KUKA KRL program: MyProgram_095().src

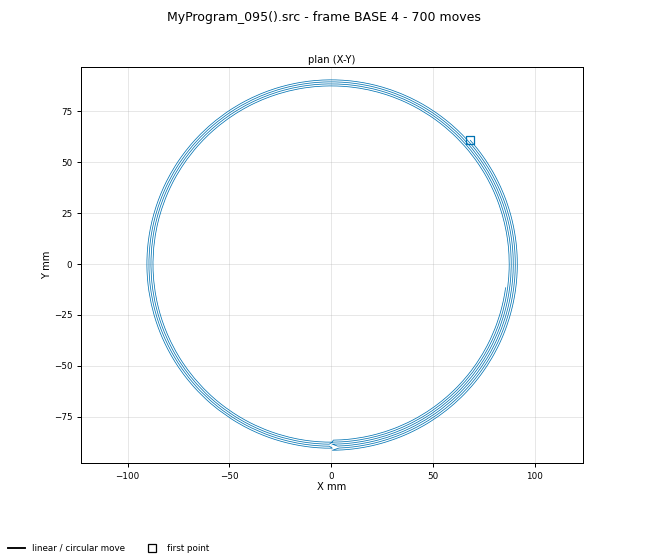
[picture p0: tool path of MyProgram_095().src in frame BASE 4, 700 of 700 moves have a stored position in this frame; points joined in program order, loops and branches not executed]
&ACCESS RVP
&REL 1
&PARAM TEMPLATE = C:\KRC\Roboter\Template\vorgabe
&PARAM EDITMASK = *
DEF MyProgram_095()
; ---- Setting reference (Base) ----
$BASE = BASE_DATA[4]

; --------------------------
; ---- Setting tool (TCP) ----
$TOOL = TOOL_DATA[3]
; --------------------------

$VEL.CP = VEL_APROX_PRINT
Startdeposition()
$VEL.CP = VEL_PRINT
LIN {X 68.4348,Y 60.7863,Z 89,A 36.1142,B 24.9115,C -2.1728,E1 25.1202,E2 408.9447} C_DIS
LIN {X 69.906,Y 59.0885,Z 89,A 34.5968,B 24.912,C -2.1656,E1 25.123,E2 410.4721} C_DIS
LIN {X 71.8852,Y 56.6631,Z 89,A 32.7208,B 24.9122,C -2.1639,E1 25.1263,E2 412.3433} C_DIS
LIN {X 73.5209,Y 54.5268,Z 89,A 31.0903,B 24.9124,C -2.1617,E1 25.129,E2 413.9712} C_DIS
LIN {X 74.8369,Y 52.7061,Z 89,A 29.6918,B 24.9126,C -2.1585,E1 25.1313,E2 415.3706} C_DIS
LIN {X 76.1078,Y 50.8536,Z 89,A 28.2935,B 24.9129,C -2.1552,E1 25.1335,E2 416.7698} C_DIS
LIN {X 77.3329,Y 48.9705,Z 89,A 26.8951,B 24.9132,C -2.1518,E1 25.1356,E2 418.169} C_DIS
LIN {X 78.5114,Y 47.0579,Z 89,A 25.4966,B 24.9134,C -2.1484,E1 25.1376,E2 419.5685} C_DIS
LIN {X 79.5405,Y 45.2947,Z 89,A 24.2263,B 24.9137,C -2.1453,E1 25.1394,E2 420.8396} C_DIS
LIN {X 80.6281,Y 43.329,Z 89,A 22.8286,B 24.914,C -2.1418,E1 25.1413,E2 422.2383} C_DIS
LIN {X 81.9545,Y 40.7633,Z 89,A 20.9127,B 24.9147,C -2.1329,E1 25.1437,E2 424.165} C_DIS
LIN {X 83.2199,Y 38.1175,Z 89,A 19.2069,B 24.9147,C -2.1324,E1 25.1457,E2 425.8628} C_DIS
LIN {X 84.1302,Y 36.0637,Z 89,A 17.8095,B 24.915,C -2.1287,E1 25.1473,E2 427.2613} C_DIS
LIN {X 84.9127,Y 34.178,Z 89,A 16.5212,B 24.9153,C -2.1247,E1 25.1486,E2 428.552} C_DIS
LIN {X 86.1131,Y 31.0294,Z 89,A 14.4253,B 24.9158,C -2.119,E1 25.1507,E2 430.6496} C_DIS
LIN {X 86.9142,Y 28.7126,Z 89,A 12.9188,B 24.9161,C -2.1154,E1 25.152,E2 432.1561} C_DIS
LIN {X 87.532,Y 26.7667,Z 89,A 11.6496,B 24.9164,C -2.1119,E1 25.1531,E2 433.4263} C_DIS
LIN {X 88.3281,Y 24.0072,Z 89,A 9.739,B 24.9171,C -2.1024,E1 25.1545,E2 435.3484} C_DIS
LIN {X 89.0572,Y 21.1497,Z 89,A 8.0298,B 24.9171,C -2.1017,E1 25.1557,E2 437.0493} C_DIS
LIN {X 89.6843,Y 18.3008,Z 89,A 6.1409,B 24.9178,C -2.0938,E1 25.1568,E2 438.9459} C_DIS
LIN {X 90.2812,Y 15.0822,Z 89,A 4.0769,B 24.9183,C -2.0868,E1 25.1578,E2 441.0142} C_DIS
LIN {X 90.6725,Y 12.5216,Z 89,A 2.552,B 24.9185,C -2.0853,E1 25.1584,E2 442.5338} C_DIS
LIN {X 90.9525,Y 10.2926,Z 89,A 1.1555,B 24.9188,C -2.0812,E1 25.1589,E2 443.9317} C_DIS
LIN {X 91.2533,Y 7.1433,Z 89,A -0.8295,B 24.9193,C -2.0747,E1 25.1594,E2 445.9201} C_DIS
LIN {X 91.4238,Y 4.4914,Z 89,A -2.4448,B 24.9196,C -2.0712,E1 25.1596,E2 447.5343} C_DIS
LIN {X 91.5002,Y 2.4512,Z 89,A -3.8938,B 24.9204,C -2.0608,E1 25.1598,E2 448.999} C_DIS
LIN {X 91.5272,Y -1.1233,Z 89,A -5.9356,B 24.9204,C -2.0608,E1 25.1598,E2 451.0288} C_DIS
LIN {X 91.4721,Y -3.3691,Z 89,A -7.3323,B 24.9207,C -2.0566,E1 25.1596,E2 452.427} C_DIS
LIN {X 91.2861,Y -6.7337,Z 89,A -9.4265,B 24.9212,C -2.0504,E1 25.1593,E2 454.5234} C_DIS
LIN {X 91.0357,Y -9.5222,Z 89,A -11.2776,B 24.9219,C -2.0412,E1 25.1588,E2 456.3854} C_DIS
LIN {X 90.7277,Y -12.1155,Z 89,A -12.8086,B 24.9219,C -2.0397,E1 25.1583,E2 457.9108} C_DIS
LIN {X 90.403,Y -14.3384,Z 89,A -14.205,B 24.9223,C -2.0356,E1 25.1577,E2 459.3087} C_DIS
LIN {X 90.0239,Y -16.5527,Z 89,A -15.583,B 24.9226,C -2.0321,E1 25.157,E2 460.6868} C_DIS
LIN {X 89.5906,Y -18.757,Z 89,A -16.9981,B 24.9229,C -2.0273,E1 25.1562,E2 462.1049} C_DIS
LIN {X 89.1033,Y -20.95,Z 89,A -18.3945,B 24.9232,C -2.0232,E1 25.1553,E2 463.503} C_DIS
LIN {X 88.3471,Y -23.9366,Z 89,A -20.3496,B 24.9238,C -2.0162,E1 25.154,E2 465.4634} C_DIS
LIN {X 87.5927,Y -26.5709,Z 89,A -21.9951,B 24.924,C -2.0133,E1 25.1527,E2 467.1063} C_DIS
LIN {X 86.9773,Y -28.5176,Z 89,A -23.2641,B 24.9243,C -2.0097,E1 25.1516,E2 468.3767} C_DIS
LIN {X 86.2512,Y -30.6435,Z 89,A -24.6609,B 24.9246,C -2.0057,E1 25.1503,E2 469.7751} C_DIS
LIN {X 85.5341,Y -32.5902,Z 89,A -26.0056,B 24.925,C -2,E1 25.149,E2 471.1257} C_DIS
LIN {X 84.6437,Y -34.8388,Z 89,A -27.4729,B 24.9252,C -1.997,E1 25.1474,E2 472.5918} C_DIS
LIN {X 83.7633,Y -36.9055,Z 89,A -28.8517,B 24.9255,C -1.9938,E1 25.1459,E2 473.9708} C_DIS
LIN {X 82.8323,Y -38.9501,Z 89,A -30.2672,B 24.9258,C -1.9892,E1 25.1442,E2 475.3893} C_DIS
LIN {X 81.7605,Y -41.1548,Z 89,A -31.9887,B 24.9267,C -1.9778,E1 25.1421,E2 477.1286} C_DIS
LIN {X 80.1903,Y -44.1362,Z 89,A -33.8687,B 24.9265,C -1.98,E1 25.1396,E2 478.9936} C_DIS
LIN {X 79.083,Y -46.0909,Z 89,A -35.2665,B 24.9268,C -1.9762,E1 25.1377,E2 480.393} C_DIS
LIN {X 77.928,Y -48.0178,Z 89,A -36.6636,B 24.927,C -1.9725,E1 25.1356,E2 481.7917} C_DIS
LIN {X 76.7342,Y -49.9032,Z 89,A -38.0524,B 24.9273,C -1.9689,E1 25.1335,E2 483.1821} C_DIS
LIN {X 75.2678,Y -52.0862,Z 89,A -39.8077,B 24.9279,C -1.9604,E1 25.1308,E2 484.9489} C_DIS
LIN {X 73.5209,Y -54.5268,Z 89,A -41.556,B 24.9279,C -1.96,E1 25.1279,E2 486.6897} C_DIS
LIN {X 72.2857,Y -56.1523,Z 89,A -42.8446,B 24.9283,C -1.9562,E1 25.1257,E2 487.9811} C_DIS
LIN {X 70.7568,Y -58.0686,Z 89,A -44.3521,B 24.9285,C -1.9531,E1 25.1231,E2 489.4889} C_DIS
LIN {X 69.3104,Y -59.7876,Z 89,A -45.7504,B 24.9287,C -1.9497,E1 25.1205,E2 490.8888} C_DIS
LIN {X 67.0628,Y -62.2982,Z 89,A -47.8483,B 24.9291,C -1.9448,E1 25.1166,E2 492.989} C_DIS
LIN {X 65.5138,Y -63.9252,Z 89,A -49.2469,B 24.9293,C -1.9416,E1 25.1139,E2 494.3892} C_DIS
LIN {X 63.9252,Y -65.5138,Z 89,A -50.6456,B 24.9295,C -1.9385,E1 25.1111,E2 495.7893} C_DIS
LIN {X 62.2982,Y -67.0628,Z 89,A -52.0445,B 24.9298,C -1.9354,E1 25.1083,E2 497.1897} C_DIS
LIN {X 60.7039,Y -68.5086,Z 89,A -53.59,B 24.9305,C -1.9252,E1 25.105,E2 498.7532} C_DIS
LIN {X 58.2262,Y -70.6258,Z 89,A -55.415,B 24.9303,C -1.9284,E1 25.1011,E2 500.5637} C_DIS
LIN {X 56.4754,Y -72.0335,Z 89,A -56.833,B 24.9305,C -1.9249,E1 25.098,E2 501.9846} C_DIS
LIN {X 54.6906,Y -73.3978,Z 89,A -58.2143,B 24.9307,C -1.9228,E1 25.0949,E2 503.3659} C_DIS
LIN {X 53.0381,Y -74.6,Z 89,A -59.5276,B 24.931,C -1.919,E1 25.092,E2 504.6836} C_DIS
LIN {X 50.8536,Y -76.1078,Z 89,A -61.142,B 24.931,C -1.9173,E1 25.0882,E2 506.2965} C_DIS
LIN {X 49.143,Y -77.2222,Z 89,A -62.4148,B 24.9312,C -1.915,E1 25.0852,E2 507.5706} C_DIS
LIN {X 47.2331,Y -78.405,Z 89,A -63.8151,B 24.9314,C -1.9126,E1 25.0819,E2 508.9721} C_DIS
LIN {X 45.2947,Y -79.5405,Z 89,A -65.2344,B 24.9316,C -1.9096,E1 25.0785,E2 510.3943} C_DIS
LIN {X 42.4309,Y -81.104,Z 89,A -67.2665,B 24.9319,C -1.9065,E1 25.0735,E2 512.428} C_DIS
LIN {X 40.332,Y -82.1683,Z 89,A -68.7183,B 24.9319,C -1.9048,E1 25.0698,E2 513.8798} C_DIS
LIN {X 38.1175,Y -83.2199,Z 89,A -70.2478,B 24.9321,C -1.9025,E1 25.066,E2 515.4108} C_DIS
LIN {X 36.0637,Y -84.1302,Z 89,A -71.6494,B 24.9323,C -1.9006,E1 25.0624,E2 516.8135} C_DIS
LIN {X 33.9882,Y -84.99,Z 89,A -73.247,B 24.9329,C -1.8919,E1 25.0582,E2 518.428} C_DIS
LIN {X 30.8369,Y -86.1834,Z 89,A -75.1546,B 24.9326,C -1.8961,E1 25.0532,E2 520.3216} C_DIS
LIN {X 28.7126,Y -86.9142,Z 89,A -76.5571,B 24.9327,C -1.8945,E1 25.0495,E2 521.7252} C_DIS
LIN {X 26.7667,Y -87.532,Z 89,A -77.8313,B 24.9328,C -1.8932,E1 25.0461,E2 523.0004} C_DIS
LIN {X 24.4133,Y -88.2184,Z 89,A -79.3626,B 24.9329,C -1.8916,E1 25.042,E2 524.5328} C_DIS
LIN {X 22.241,Y -88.7909,Z 89,A -80.7653,B 24.933,C -1.8903,E1 25.0382,E2 525.9364} C_DIS
LIN {X 20.0552,Y -89.31,Z 89,A -82.1687,B 24.9331,C -1.889,E1 25.0344,E2 527.3409} C_DIS
LIN {X 17.8574,Y -89.7753,Z 89,A -83.5725,B 24.9331,C -1.8879,E1 25.0305,E2 528.7457} C_DIS
LIN {X 15.6488,Y -90.1865,Z 89,A -85.1605,B 24.9337,C -1.8806,E1 25.0261,E2 530.3492} C_DIS
LIN {X 12.5216,Y -90.6725,Z 89,A -86.9727,B 24.9334,C -1.8849,E1 25.0212,E2 532.1494} C_DIS
LIN {X 10.2926,Y -90.9525,Z 89,A -88.377,B 24.9334,C -1.8841,E1 25.0173,E2 533.5545} C_DIS
LIN {X 8.0575,Y -91.1777,Z 89,A -89.7817,B 24.9335,C -1.8835,E1 25.0134,E2 534.9601} C_DIS
LIN {X 5.8174,Y -91.348,Z 89,A -91.1865,B 24.9335,C -1.8829,E1 25.0094,E2 536.3656} C_DIS
LIN {X 2.5555,Y -91.497,Z 89,A -93.2493,B 24.9336,C -1.8815,E1 25.0037,E2 538.4311} C_DIS
LIN {X 0.6147,Y -91.5303,Z 89,A -94.1302,B 24.9329,C -1.8925,E1 25.0013,E2 539.2859} C_DIS
Enddeposition()
LIN {X 0.6147,Y -91.5303,Z 89,A -94.1302,B 24.9329,C -1.8925,E1 25.0013,E2 539.2859} C_DIS
Startdeposition()
$VEL.CP = VEL_PRINT
LIN {X 3.841,Y -90.4576,Z 89,A -91.6476,B 24.9305,C -1.9253,E1 25.0084,E2 536.7259} C_DIS
LIN {X 6.8274,Y -90.2822,Z 89,A -89.6587,B 24.9302,C -1.9294,E1 25.014,E2 534.7283} C_DIS
LIN {X 10.5822,Y -89.9186,Z 89,A -87.3173,B 24.9302,C -1.9292,E1 25.0205,E2 532.3889} C_DIS
LIN {X 13.8939,Y -89.4668,Z 89,A -84.9684,B 24.9295,C -1.9387,E1 25.027,E2 530.0197} C_DIS
LIN {X 18.0628,Y -88.7192,Z 89,A -82.5559,B 24.93,C -1.9317,E1 25.0336,E2 527.6266} C_DIS
LIN {X 21.585,Y -87.9286,Z 89,A -80.3322,B 24.93,C -1.9317,E1 25.0397,E2 525.4058} C_DIS
LIN {X 23.7624,Y -87.3654,Z 89,A -78.7831,B 24.9296,C -1.9376,E1 25.0439,E2 523.8453} C_DIS
LIN {X 27.8255,Y -86.1573,Z 89,A -75.9416,B 24.929,C -1.9463,E1 25.0515,E2 520.9884} C_DIS
LIN {X 32.3644,Y -84.5576,Z 89,A -72.9807,B 24.929,C -1.9473,E1 25.0592,E2 518.0312} C_DIS
LIN {X 36.0562,Y -83.05,Z 89,A -70.5763,B 24.929,C -1.9468,E1 25.0654,E2 515.6336} C_DIS
LIN {X 39.4601,Y -81.4881,Z 89,A -68.247,B 24.9288,C -1.9491,E1 25.0713,E2 513.3049} C_DIS
LIN {X 42.1763,Y -80.1155,Z 89,A -65.821,B 24.9272,C -1.9701,E1 25.0774,E2 510.8361} C_DIS
LIN {X 45.1686,Y -78.4674,Z 89,A -64.2021,B 24.9284,C -1.9546,E1 25.0812,E2 509.2585} C_DIS
LIN {X 48.0241,Y -76.753,Z 89,A -61.7848,B 24.9273,C -1.9696,E1 25.087,E2 506.8135} C_DIS
LIN {X 51.7728,Y -74.276,Z 89,A -59.1835,B 24.9275,C -1.9666,E1 25.093,E2 504.2281} C_DIS
LIN {X 53.7404,Y -72.8657,Z 89,A -57.2283,B 24.9261,C -1.985,E1 25.0975,E2 502.2365} C_DIS
LIN {X 56.4119,Y -70.8178,Z 89,A -55.1326,B 24.9259,C -1.9884,E1 25.102,E2 500.1406} C_DIS
LIN {X 58.9229,Y -68.7422,Z 89,A -53.6408,B 24.9271,C -1.9725,E1 25.1051,E2 498.6921} C_DIS
LIN {X 60.8149,Y -67.075,Z 89,A -51.7631,B 24.926,C -1.9863,E1 25.1091,E2 496.7893} C_DIS
LIN {X 63.9525,Y -64.0907,Z 89,A -49.1215,B 24.9258,C -1.9893,E1 25.1144,E2 494.1516} C_DIS
LIN {X 66.8951,Y -61.0119,Z 89,A -46.6842,B 24.926,C -1.9867,E1 25.119,E2 491.7311} C_DIS
LIN {X 68.7114,Y -58.9592,Z 89,A -44.8258,B 24.9253,C -1.9957,E1 25.1224,E2 489.86} C_DIS
LIN {X 70.8722,Y -56.343,Z 89,A -42.7154,B 24.925,C -2,E1 25.1261,E2 487.7491} C_DIS
LIN {X 72.9495,Y -53.6259,Z 89,A -40.3766,B 24.9241,C -2.0122,E1 25.1301,E2 485.3927} C_DIS
LIN {X 74.6947,Y -51.1692,Z 89,A -38.0119,B 24.9224,C -2.0342,E1 25.1339,E2 482.9877} C_DIS
LIN {X 76.7688,Y -47.9989,Z 89,A -36.3079,B 24.9238,C -2.0156,E1 25.1363,E2 481.3363} C_DIS
LIN {X 78.8273,Y -44.5399,Z 89,A -33.7021,B 24.9231,C -2.025,E1 25.14,E2 478.7215} C_DIS
LIN {X 80.3925,Y -41.6488,Z 89,A -31.6323,B 24.9227,C -2.0308,E1 25.1427,E2 476.6491} C_DIS
LIN {X 81.849,Y -38.7087,Z 89,A -29.5508,B 24.9222,C -2.0371,E1 25.1452,E2 474.5638} C_DIS
LIN {X 83.2517,Y -35.5907,Z 89,A -27.6678,B 24.9225,C -2.0334,E1 25.1473,E2 472.6998} C_DIS
LIN {X 84.5175,Y -32.4701,Z 89,A -25.045,B 24.9206,C -2.058,E1 25.15,E2 470.0335} C_DIS
LIN {X 85.8563,Y -28.7415,Z 89,A -22.8423,B 24.9208,C -2.0546,E1 25.152,E2 467.8513} C_DIS
LIN {X 86.8313,Y -25.645,Z 89,A -20.7763,B 24.9203,C -2.0614,E1 25.1537,E2 465.7809} C_DIS
LIN {X 87.7136,Y -22.4425,Z 89,A -18.7465,B 24.92,C -2.0654,E1 25.1552,E2 463.7534} C_DIS
LIN {X 88.4899,Y -19.1544,Z 89,A -16.7256,B 24.9198,C -2.0679,E1 25.1564,E2 461.7384} C_DIS
LIN {X 89.1025,Y -16.0649,Z 89,A -14.6764,B 24.9192,C -2.0763,E1 25.1575,E2 459.6813} C_DIS
LIN {X 89.7875,Y -11.642,Z 89,A -11.4066,B 24.9172,C -2.1015,E1 25.1588,E2 456.3713} C_DIS
LIN {X 90.2839,Y -6.8065,Z 89,A -8.9059,B 24.9181,C -2.0901,E1 25.1594,E2 453.9122} C_DIS
LIN {X 90.4532,Y -3.9434,Z 89,A -7.0295,B 24.9174,C -2.0982,E1 25.1597,E2 452.0278} C_DIS
LIN {X 90.5369,Y -0.7324,Z 89,A -4.9658,B 24.9168,C -2.1059,E1 25.1597,E2 449.9584} C_DIS
LIN {X 90.4983,Y 2.7184,Z 89,A -2.7827,B 24.9163,C -2.1129,E1 25.1597,E2 447.7718} C_DIS
LIN {X 90.3216,Y 6.2745,Z 89,A -0.5065,B 24.9156,C -2.1209,E1 25.1593,E2 445.4902} C_DIS
LIN {X 90.012,Y 9.7618,Z 89,A 1.5203,B 24.9156,C -2.1209,E1 25.1587,E2 443.4751} C_DIS
LIN {X 89.7383,Y 12.0216,Z 89,A 3.2086,B 24.9145,C -2.1346,E1 25.1581,E2 441.7648} C_DIS
LIN {X 89.1963,Y 15.5434,Z 89,A 5.1496,B 24.9149,C -2.1301,E1 25.1573,E2 439.8457} C_DIS
LIN {X 88.7451,Y 17.9364,Z 89,A 6.8451,B 24.9141,C -2.1406,E1 25.1563,E2 438.1354} C_DIS
LIN {X 88.0369,Y 21.141,Z 89,A 8.9727,B 24.9134,C -2.1488,E1 25.155,E2 436.0007} C_DIS
LIN {X 87.4365,Y 23.4992,Z 89,A 10.4329,B 24.9133,C -2.1506,E1 25.154,E2 434.5447} C_DIS
LIN {X 85.8607,Y 28.7284,Z 89,A 13.9051,B 24.9124,C -2.1615,E1 25.1511,E2 431.0665} C_DIS
LIN {X 84.6865,Y 32.024,Z 89,A 15.7904,B 24.9128,C -2.1561,E1 25.1493,E2 429.2045} C_DIS
LIN {X 83.1699,Y 35.7813,Z 89,A 18.5222,B 24.9117,C -2.1695,E1 25.1464,E2 426.4561} C_DIS
LIN {X 82.0179,Y 38.3461,Z 89,A 20.4762,B 24.9108,C -2.1809,E1 25.1441,E2 424.4859} C_DIS
LIN {X 80.8031,Y 40.8455,Z 89,A 22.4831,B 24.9096,C -2.1947,E1 25.1416,E2 422.4569} C_DIS
LIN {X 78.9088,Y 44.3939,Z 89,A 24.6853,B 24.9101,C -2.1892,E1 25.1386,E2 420.2793} C_DIS
LIN {X 77.2267,Y 47.2594,Z 89,A 26.4874,B 24.9105,C -2.184,E1 25.1361,E2 418.4987} C_DIS
LIN {X 75.5281,Y 49.9285,Z 89,A 28.8052,B 24.9092,C -2.2004,E1 25.1325,E2 416.1537} C_DIS
LIN {X 73.3795,Y 53.0386,Z 89,A 31.4469,B 24.9079,C -2.2153,E1 25.1282,E2 413.4897} C_DIS
LIN {X 70.8403,Y 56.3833,Z 89,A 33.677,B 24.9087,C -2.2065,E1 25.1244,E2 411.2911} C_DIS
LIN {X 69.0223,Y 58.5942,Z 89,A 35.5338,B 24.9082,C -2.2123,E1 25.1211,E2 409.4289} C_DIS
LIN {X 66.3294,Y 61.6273,Z 89,A 37.9615,B 24.9082,C -2.2131,E1 25.1166,E2 407.0102} C_DIS
LIN {X 64.3928,Y 63.6467,Z 89,A 39.855,B 24.9074,C -2.2213,E1 25.1129,E2 405.1055} C_DIS
LIN {X 61.9374,Y 66.0387,Z 89,A 41.718,B 24.908,C -2.215,E1 25.1092,E2 403.265} C_DIS
LIN {X 59.5402,Y 68.2078,Z 89,A 44.0276,B 24.9069,C -2.2283,E1 25.1043,E2 400.9333} C_DIS
LIN {X 57.492,Y 69.9446,Z 89,A 45.8102,B 24.9063,C -2.2344,E1 25.1005,E2 399.1431} C_DIS
LIN {X 54.2039,Y 72.5212,Z 89,A 48.5095,B 24.9058,C -2.2411,E1 25.0945,E2 396.4377} C_DIS
LIN {X 51.4181,Y 74.5226,Z 89,A 50.2979,B 24.9066,C -2.2315,E1 25.0905,E2 394.6783} C_DIS
LIN {X 47.9538,Y 76.797,Z 89,A 53.2119,B 24.9054,C -2.2457,E1 25.0836,E2 391.7403} C_DIS
LIN {X 45.0435,Y 78.5393,Z 89,A 55.3345,B 24.9052,C -2.2479,E1 25.0785,E2 389.6188} C_DIS
LIN {X 42.687,Y 79.8461,Z 89,A 57.3502,B 24.9041,C -2.2609,E1 25.0735,E2 387.578} C_DIS
LIN {X 38.919,Y 81.7481,Z 89,A 59.8208,B 24.9044,C -2.2573,E1 25.0673,E2 385.1226} C_DIS
LIN {X 34.2257,Y 83.8209,Z 89,A 63.3531,B 24.9033,C -2.2706,E1 25.0582,E2 381.5673} C_DIS
LIN {X 29.4174,Y 85.6284,Z 89,A 66.5241,B 24.9033,C -2.2707,E1 25.0499,E2 378.4024} C_DIS
LIN {X 25.2199,Y 86.957,Z 89,A 69.0295,B 24.9039,C -2.2632,E1 25.0432,E2 375.9192} C_DIS
LIN {X 21.9677,Y 87.8352,Z 89,A 71.1397,B 24.9039,C -2.2638,E1 25.0375,E2 373.8109} C_DIS
LIN {X 18.9594,Y 88.5324,Z 89,A 72.9796,B 24.9041,C -2.261,E1 25.0325,E2 371.9801} C_DIS
LIN {X 15.891,Y 89.1338,Z 89,A 75.0794,B 24.9037,C -2.2658,E1 25.0267,E2 369.8712} C_DIS
LIN {X 12.4524,Y 89.6792,Z 89,A 77.0943,B 24.9042,C -2.2602,E1 25.0212,E2 367.8716} C_DIS
LIN {X 9.4502,Y 90.0446,Z 89,A 79.136,B 24.9038,C -2.2647,E1 25.0155,E2 365.8206} C_DIS
LIN {X 5.8559,Y 90.3499,Z 89,A 81.4804,B 24.9036,C -2.2669,E1 25.009,E2 363.4722} C_DIS
LIN {X 2.2826,Y 90.5117,Z 89,A 83.5521,B 24.9042,C -2.2604,E1 25.0033,E2 361.4165} C_DIS
LIN {X -0.6869,Y 90.5366,Z 89,A 85.6422,B 24.9036,C -2.2669,E1 24.9974,E2 359.3109} C_DIS
LIN {X -4.2126,Y 90.4417,Z 89,A 87.8996,B 24.9036,C -2.267,E1 24.9911,E2 357.0528} C_DIS
LIN {X -7.9472,Y 90.1905,Z 89,A 90.2515,B 24.9037,C -2.2654,E1 24.9845,E2 354.7037} C_DIS
LIN {X -11.1573,Y 89.8503,Z 89,A 92.3303,B 24.9037,C -2.2654,E1 24.9788,E2 352.6236} C_DIS
LIN {X -14.8513,Y 89.3128,Z 89,A 94.5753,B 24.9042,C -2.2601,E1 24.9726,E2 350.3893} C_DIS
LIN {X -17.601,Y 88.8122,Z 89,A 96.6821,B 24.9034,C -2.2695,E1 24.9668,E2 348.2577} C_DIS
LIN {X -21.5979,Y 87.9255,Z 89,A 99.0047,B 24.9043,C -2.2585,E1 24.9605,E2 345.9582} C_DIS
LIN {X -24.8007,Y 87.0763,Z 89,A 100.9732,B 24.9048,C -2.2523,E1 24.9552,E2 344.0015} C_DIS
LIN {X -27.4177,Y 86.2893,Z 89,A 102.8866,B 24.9045,C -2.2561,E1 24.9501,E2 342.0756} C_DIS
LIN {X -31.1882,Y 84.998,Z 89,A 105.4157,B 24.9048,C -2.2532,E1 24.9435,E2 339.5484} C_DIS
LIN {X -34.5944,Y 83.6708,Z 89,A 107.5352,B 24.9055,C -2.2439,E1 24.938,E2 337.4465} C_DIS
LIN {X -38.8381,Y 81.787,Z 89,A 110.6816,B 24.9054,C -2.246,E1 24.93,E2 334.2873} C_DIS
LIN {X -41.879,Y 80.2721,Z 89,A 112.7855,B 24.9058,C -2.2411,E1 24.9248,E2 332.1895} C_DIS
LIN {X -44.5871,Y 78.8009,Z 89,A 115.1067,B 24.9051,C -2.2493,E1 24.919,E2 329.842} C_DIS
LIN {X -48.6235,Y 76.3754,Z 89,A 117.709,B 24.9065,C -2.232,E1 24.9129,E2 327.2727} C_DIS
LIN {X -51.4688,Y 74.4874,Z 89,A 119.8592,B 24.9069,C -2.2275,E1 24.908,E2 325.1262} C_DIS
LIN {X -56.755,Y 70.543,Z 89,A 124.383,B 24.9068,C -2.2294,E1 24.8979,E2 320.5812} C_DIS
LIN {X -60.1524,Y 67.6692,Z 89,A 126.781,B 24.9084,C -2.2103,E1 24.8929,E2 318.2195} C_DIS
LIN {X -64.183,Y 63.8591,Z 89,A 130.3958,B 24.9088,C -2.2052,E1 24.8856,E2 314.6018} C_DIS
LIN {X -66.9222,Y 60.9824,Z 89,A 132.9651,B 24.9092,C -2.2007,E1 24.8807,E2 312.032} C_DIS
LIN {X -69.0691,Y 58.5393,Z 89,A 135.7258,B 24.9078,C -2.2168,E1 24.8756,E2 309.2202} C_DIS
LIN {X -71.5763,Y 55.4457,Z 89,A 137.5885,B 24.91,C -2.1902,E1 24.8725,E2 307.4124} C_DIS
LIN {X -73.5936,Y 52.7385,Z 89,A 139.6955,B 24.9106,C -2.1835,E1 24.8691,E2 305.311} C_DIS
LIN {X -75.3144,Y 50.2526,Z 89,A 141.7065,B 24.9108,C -2.1811,E1 24.8659,E2 303.2956} C_DIS
LIN {X -76.5996,Y 48.2697,Z 89,A 143.2253,B 24.9111,C -2.1777,E1 24.8636,E2 301.7774} C_DIS
LIN {X -78.7995,Y 44.5894,Z 89,A 146.1309,B 24.9112,C -2.1757,E1 24.8595,E2 298.8615} C_DIS
LIN {X -80.8397,Y 40.7739,Z 89,A 148.829,B 24.912,C -2.1664,E1 24.8561,E2 296.171} C_DIS
LIN {X -82.3206,Y 37.6953,Z 89,A 150.9163,B 24.9127,C -2.1577,E1 24.8536,E2 294.0931} C_DIS
LIN {X -83.798,Y 34.282,Z 89,A 153.1681,B 24.9135,C -2.1476,E1 24.8512,E2 291.8531} C_DIS
LIN {X -84.9131,Y 31.4209,Z 89,A 155.6055,B 24.9128,C -2.1564,E1 24.8488,E2 289.3807} C_DIS
LIN {X -85.9862,Y 28.3543,Z 89,A 157.9259,B 24.9127,C -2.158,E1 24.8468,E2 287.0433} C_DIS
LIN {X -87.1572,Y 24.5149,Z 89,A 159.6948,B 24.9152,C -2.1269,E1 24.8455,E2 285.3383} C_DIS
LIN {X -88.0666,Y 21.0193,Z 89,A 162.16,B 24.9153,C -2.1251,E1 24.8438,E2 282.8632} C_DIS
LIN {X -88.8209,Y 17.5612,Z 89,A 164.3658,B 24.916,C -2.1169,E1 24.8425,E2 280.6638} C_DIS
LIN {X -89.4048,Y 14.2946,Z 89,A 166.4804,B 24.9164,C -2.1107,E1 24.8416,E2 278.5516} C_DIS
LIN {X -89.8714,Y 10.9855,Z 89,A 168.3538,B 24.9176,C -2.0968,E1 24.8409,E2 276.7003} C_DIS
LIN {X -90.1183,Y 8.7287,Z 89,A 170.0477,B 24.9173,C -2.0998,E1 24.8404,E2 274.9889} C_DIS
LIN {X -90.3804,Y 5.3726,Z 89,A 172.1787,B 24.9178,C -2.093,E1 24.84,E2 272.8614} C_DIS
LIN {X -90.5176,Y 2.0025,Z 89,A 174.2642,B 24.9185,C -2.0847,E1 24.8398,E2 270.7831} C_DIS
LIN {X -90.5355,Y -0.9214,Z 89,A 176.0887,B 24.919,C -2.078,E1 24.8398,E2 268.9636} C_DIS
LIN {X -90.4602,Y -3.782,Z 89,A 177.956,B 24.9193,C -2.0739,E1 24.84,E2 267.0948} C_DIS
LIN {X -90.2522,Y -7.203,Z 89,A -179.8808,B 24.9199,C -2.0669,E1 24.8404,E2 264.9354} C_DIS
LIN {X -89.937,Y -10.4248,Z 89,A -178.1412,B 24.9211,C -2.0512,E1 24.8409,E2 263.2227} C_DIS
LIN {X -89.5869,Y -13.102,Z 89,A -176.1167,B 24.9208,C -2.0552,E1 24.8417,E2 261.1765} C_DIS
LIN {X -88.3611,Y -19.7448,Z 89,A -171.9405,B 24.922,C -2.039,E1 24.8439,E2 257.0145} C_DIS
LIN {X -86.9694,Y -25.1777,Z 89,A -168.234,B 24.9225,C -2.0328,E1 24.8465,E2 253.3011} C_DIS
LIN {X -86.0678,Y -28.1022,Z 89,A -166.2597,B 24.9229,C -2.0282,E1 24.8482,E2 251.3265} C_DIS
LIN {X -85.0374,Y -31.0801,Z 89,A -164.352,B 24.9235,C -2.0197,E1 24.8499,E2 249.4282} C_DIS
LIN {X -84.02,Y -33.7367,Z 89,A -162.5395,B 24.9239,C -2.0149,E1 24.8518,E2 247.6171} C_DIS
LIN {X -82.9012,Y -36.3975,Z 89,A -160.4792,B 24.9237,C -2.0167,E1 24.8541,E2 245.5409} C_DIS
LIN {X -81.6835,Y -39.0534,Z 89,A -158.7203,B 24.9243,C -2.0088,E1 24.8561,E2 243.7913} C_DIS
LIN {X -80.2825,Y -41.8592,Z 89,A -156.6185,B 24.9245,C -2.0069,E1 24.8588,E2 241.6828} C_DIS
LIN {X -78.6247,Y -44.895,Z 89,A -154.4844,B 24.925,C -1.9994,E1 24.8617,E2 239.5555} C_DIS
LIN {X -76.7901,Y -47.9648,Z 89,A -152.2371,B 24.9255,C -1.993,E1 24.865,E2 237.3119} C_DIS
LIN {X -74.9211,Y -50.8347,Z 89,A -150.2206,B 24.9263,C -1.9829,E1 24.8681,E2 235.3095} C_DIS
LIN {X -72.5165,Y -54.2101,Z 89,A -146.9092,B 24.9252,C -1.9977,E1 24.8736,E2 231.9468} C_DIS
LIN {X -70.4943,Y -56.815,Z 89,A -144.8961,B 24.9257,C -1.9904,E1 24.8771,E2 229.9415} C_DIS
LIN {X -67.4946,Y -60.3475,Z 89,A -142.4087,B 24.9272,C -1.97,E1 24.8816,E2 227.4916} C_DIS
LIN {X -65.4359,Y -62.5748,Z 89,A -140.4813,B 24.9275,C -1.966,E1 24.8853,E2 225.5653} C_DIS
LIN {X -61.199,Y -66.7234,Z 89,A -136.6314,B 24.9279,C -1.9613,E1 24.8931,E2 221.7105} C_DIS
LIN {X -59.1444,Y -68.5534,Z 89,A -134.4581,B 24.9271,C -1.9715,E1 24.8977,E2 219.5044} C_DIS
LIN {X -55.3298,Y -71.6656,Z 89,A -131.7208,B 24.9284,C -1.9539,E1 24.9036,E2 216.7989} C_DIS
LIN {X -48.8404,Y -76.2362,Z 89,A -126.6847,B 24.929,C -1.9461,E1 24.9152,E2 211.7644} C_DIS
LIN {X -46.7806,Y -77.5177,Z 89,A -124.8121,B 24.9284,C -1.9546,E1 24.9198,E2 209.8657} C_DIS
LIN {X -42.7011,Y -79.8388,Z 89,A -122.1288,B 24.9293,C -1.9414,E1 24.9263,E2 207.2063} C_DIS
LIN {X -39.6053,Y -81.4183,Z 89,A -119.4296,B 24.9283,C -1.9549,E1 24.9331,E2 204.4678} C_DIS
LIN {X -36.3709,Y -82.9128,Z 89,A -117.2406,B 24.9287,C -1.9503,E1 24.9387,E2 202.2844} C_DIS
LIN {X -33.2705,Y -84.2048,Z 89,A -115.9269,B 24.9308,C -1.9219,E1 24.9419,E2 201.0356} C_DIS
LIN {X -30.2052,Y -85.3524,Z 89,A -113.7224,B 24.9306,C -1.9243,E1 24.9477,E2 198.8208} C_DIS
LIN {X -27.7315,Y -86.1877,Z 89,A -111.9056,B 24.9303,C -1.9284,E1 24.9526,E2 196.9909} C_DIS
LIN {X -24.3899,Y -87.1927,Z 89,A -109.7191,B 24.9304,C -1.9262,E1 24.9584,E2 194.8062} C_DIS
LIN {X -21.3701,Y -87.981,Z 89,A -107.8083,B 24.9307,C -1.923,E1 24.9636,E2 192.9002} C_DIS
LIN {X -18.2981,Y -88.6709,Z 89,A -105.7306,B 24.9305,C -1.9249,E1 24.9693,E2 190.8154} C_DIS
LIN {X -15.4393,Y -89.2145,Z 89,A -103.7915,B 24.9304,C -1.9275,E1 24.9747,E2 188.8682} C_DIS
LIN {X -12.0071,Y -89.7402,Z 89,A -101.8998,B 24.9311,C -1.9168,E1 24.9798,E2 187.0002} C_DIS
LIN {X -9.9221,Y -89.9952,Z 89,A -100.2128,B 24.9303,C -1.9285,E1 24.9846,E2 185.2842} C_DIS
LIN {X -6.5554,Y -90.3026,Z 89,A -98.1699,B 24.9305,C -1.9253,E1 24.9902,E2 183.2482} C_DIS
LIN {X -3.0532,Y -90.4881,Z 89,A -95.9604,B 24.9305,C -1.9251,E1 24.9964,E2 181.0386} C_DIS
LIN {X 0.5983,Y -90.5098,Z 89,A -93.6411,B 24.9305,C -1.9264,E1 25.0029,E2 178.7164} C_DIS
Enddeposition()
LIN {X 0.5983,Y -90.5098,Z 89,A -93.6411,B 24.9305,C -1.9264,E1 25.0029,E2 178.7164} C_DIS
Startdeposition()
$VEL.CP = VEL_PRINT
LIN {X -0.8087,Y -89.5426,Z 89,A -95.5328,B 24.9316,C -1.91,E1 24.9975,E2 180.6469} C_DIS
LIN {X -3.833,Y -89.4638,Z 89,A -97.4446,B 24.9316,C -1.9105,E1 24.9922,E2 182.5577} C_DIS
LIN {X -7.8248,Y -89.2043,Z 89,A -99.8128,B 24.9311,C -1.9168,E1 24.9856,E2 184.9121} C_DIS
LIN {X -9.959,Y -88.9916,Z 89,A -101.4588,B 24.9318,C -1.908,E1 24.981,E2 186.5797} C_DIS
LIN {X -13.1443,Y -88.5776,Z 89,A -103.4787,B 24.9316,C -1.9096,E1 24.9754,E2 188.5975} C_DIS
LIN {X -16.5758,Y -87.9991,Z 89,A -105.6338,B 24.9314,C -1.9126,E1 24.9695,E2 190.7476} C_DIS
LIN {X -21.0253,Y -87.0428,Z 89,A -108.2936,B 24.9307,C -1.9221,E1 24.9623,E2 193.3882} C_DIS
LIN {X -23.2406,Y -86.4775,Z 89,A -110.1266,B 24.9315,C -1.9111,E1 24.9573,E2 195.25} C_DIS
LIN {X -26.5621,Y -85.5156,Z 89,A -112.3359,B 24.9315,C -1.9128,E1 24.9513,E2 197.4591} C_DIS
LIN {X -29.1448,Y -84.6713,Z 89,A -114.2107,B 24.9316,C -1.9099,E1 24.9464,E2 199.3443} C_DIS
LIN {X -32.5202,Y -83.4324,Z 89,A -116.4859,B 24.9314,C -1.9128,E1 24.9404,E2 201.6174} C_DIS
LIN {X -38.8769,Y -80.6664,Z 89,A -120.6985,B 24.9306,C -1.9246,E1 24.9297,E2 205.8119} C_DIS
LIN {X -42.1472,Y -79.0083,Z 89,A -123.0786,B 24.9304,C -1.9265,E1 24.9238,E2 208.1941} C_DIS
LIN {X -45.8339,Y -76.9274,Z 89,A -125.7274,B 24.93,C -1.9322,E1 24.9174,E2 210.8372} C_DIS
LIN {X -48.6331,Y -75.1883,Z 89,A -129.1049,B 24.9326,C -1.8967,E1 24.9093,E2 214.31} C_DIS
LIN {X -53.0597,Y -72.133,Z 89,A -131.4149,B 24.9297,C -1.9368,E1 24.9042,E2 216.5327} C_DIS
LIN {X -55.6777,Y -70.1321,Z 89,A -134.0228,B 24.9305,C -1.9254,E1 24.8984,E2 219.1773} C_DIS
LIN {X -59.1524,Y -67.2278,Z 89,A -136.7218,B 24.9297,C -1.937,E1 24.8928,E2 221.8593} C_DIS
LIN {X -64.2591,Y -62.3646,Z 89,A -140.8565,B 24.9281,C -1.9577,E1 24.8845,E2 225.9619} C_DIS
LIN {X -66.1025,Y -60.4067,Z 89,A -142.88,B 24.9285,C -1.9524,E1 24.8807,E2 228.007} C_DIS
LIN {X -69.567,Y -56.3818,Z 89,A -146.2048,B 24.9278,C -1.9624,E1 24.8747,E2 231.3231} C_DIS
LIN {X -73.1126,Y -51.7026,Z 89,A -150.1253,B 24.9275,C -1.9667,E1 24.8682,E2 235.2524} C_DIS
LIN {X -75.351,Y -48.3808,Z 89,A -152.44,B 24.9265,C -1.9806,E1 24.8646,E2 237.5455} C_DIS
LIN {X -76.967,Y -45.7669,Z 89,A -154.451,B 24.9262,C -1.9844,E1 24.8617,E2 239.5577} C_DIS
LIN {X -78.4752,Y -43.132,Z 89,A -156.7749,B 24.9266,C -1.9784,E1 24.8585,E2 241.9082} C_DIS
LIN {X -80.1693,Y -39.892,Z 89,A -158.7835,B 24.9254,C -1.9945,E1 24.856,E2 243.8891} C_DIS
LIN {X -81.9059,Y -36.1953,Z 89,A -161.5351,B 24.9252,C -1.9978,E1 24.8528,E2 246.6478} C_DIS
LIN {X -83.283,Y -32.9006,Z 89,A -163.7117,B 24.9244,C -2.0076,E1 24.8505,E2 248.8133} C_DIS
LIN {X -84.5299,Y -29.5497,Z 89,A -165.9304,B 24.9238,C -2.0163,E1 24.8484,E2 251.0237} C_DIS
LIN {X -85.5413,Y -26.4793,Z 89,A -168.0336,B 24.9234,C -2.0214,E1 24.8466,E2 253.1267} C_DIS
LIN {X -86.8668,Y -21.7438,Z 89,A -171.1445,B 24.9226,C -2.032,E1 24.8444,E2 256.2305} C_DIS
LIN {X -87.4063,Y -19.4618,Z 89,A -173.208,B 24.9235,C -2.0203,E1 24.8431,E2 258.334} C_DIS
LIN {X -88.4082,Y -14.2389,Z 89,A -176.0427,B 24.9214,C -2.0473,E1 24.8417,E2 261.1212} C_DIS
LIN {X -88.9734,Y -10.1144,Z 89,A -178.8916,B 24.9212,C -2.0503,E1 24.8407,E2 263.9799} C_DIS
LIN {X -89.2797,Y -6.9039,Z 89,A 178.9861,B 24.9208,C -2.0551,E1 24.8402,E2 266.1034} C_DIS
LIN {X -89.5094,Y -2.5637,Z 89,A 175.8146,B 24.921,C -2.0528,E1 24.8398,E2 269.2996} C_DIS
LIN {X -89.5218,Y 2.1368,Z 89,A 173.0982,B 24.9196,C -2.0707,E1 24.8398,E2 271.9894} C_DIS
LIN {X -89.2389,Y 7.4143,Z 89,A 169.9559,B 24.9182,C -2.0885,E1 24.8404,E2 275.1083} C_DIS
LIN {X -88.7822,Y 11.6713,Z 89,A 167.1916,B 24.9176,C -2.0965,E1 24.8413,E2 277.87} C_DIS
LIN {X -88.4062,Y 14.2508,Z 89,A 165.3153,B 24.9176,C -2.0958,E1 24.8421,E2 279.7591} C_DIS
LIN {X -87.8309,Y 17.4495,Z 89,A 163.0946,B 24.9174,C -2.0984,E1 24.8433,E2 281.9869} C_DIS
LIN {X -87.2592,Y 20.1074,Z 89,A 161.1773,B 24.9174,C -2.0988,E1 24.8445,E2 283.9144} C_DIS
LIN {X -86.3537,Y 23.6989,Z 89,A 158.9208,B 24.9165,C -2.1095,E1 24.8461,E2 286.1586} C_DIS
LIN {X -85.0126,Y 28.1352,Z 89,A 156.042,B 24.9156,C -2.1212,E1 24.8485,E2 289.026} C_DIS
LIN {X -83.4398,Y 32.5014,Z 89,A 153.4806,B 24.9139,C -2.1421,E1 24.8509,E2 291.5519} C_DIS
LIN {X -82.6252,Y 34.52,Z 89,A 151.7782,B 24.9143,C -2.1373,E1 24.8527,E2 293.2751} C_DIS
LIN {X -81.4377,Y 37.2368,Z 89,A 149.8234,B 24.914,C -2.1414,E1 24.855,E2 295.2311} C_DIS
LIN {X -80.2622,Y 39.7045,Z 89,A 148.1057,B 24.9135,C -2.1475,E1 24.8571,E2 296.9435} C_DIS
LIN {X -77.4532,Y 44.9401,Z 89,A 144.7361,B 24.9116,C -2.1711,E1 24.8615,E2 300.2746} C_DIS
LIN {X -75.2592,Y 48.5239,Z 89,A 142.0119,B 24.9111,C -2.1776,E1 24.8655,E2 302.9972} C_DIS
LIN {X -74.0661,Y 50.326,Z 89,A 140.0806,B 24.9121,C -2.1654,E1 24.8685,E2 304.9673} C_DIS
LIN {X -71.2884,Y 54.1912,Z 89,A 136.9708,B 24.9115,C -2.1717,E1 24.8737,E2 308.0771} C_DIS
LIN {X -68.2323,Y 57.99,Z 89,A 134.3702,B 24.9096,C -2.1951,E1 24.8782,E2 310.6339} C_DIS
LIN {X -66.6414,Y 59.8114,Z 89,A 132.1352,B 24.911,C -2.1787,E1 24.8824,E2 312.9179} C_DIS
LIN {X -64.1941,Y 62.4319,Z 89,A 130.2535,B 24.9095,C -2.1965,E1 24.8859,E2 314.7655} C_DIS
LIN {X -60.6838,Y 65.8482,Z 89,A 127.2519,B 24.9086,C -2.2078,E1 24.892,E2 317.7525} C_DIS
LIN {X -58.7329,Y 67.5941,Z 89,A 125.1869,B 24.9092,C -2.2,E1 24.8963,E2 319.8443} C_DIS
LIN {X -56.2455,Y 69.6775,Z 89,A 123.082,B 24.9089,C -2.2037,E1 24.9009,E2 321.9484} C_DIS
LIN {X -51.9895,Y 72.9079,Z 89,A 120.2304,B 24.9069,C -2.2278,E1 24.9071,E2 324.7529} C_DIS
LIN {X -50.2161,Y 74.1405,Z 89,A 118.3679,B 24.9079,C -2.216,E1 24.9115,E2 326.6497} C_DIS
LIN {X -46.8708,Y 76.3006,Z 89,A 115.2256,B 24.909,C -2.203,E1 24.919,E2 329.8329} C_DIS
LIN {X -43.8869,Y 78.0543,Z 89,A 113.534,B 24.9073,C -2.2226,E1 24.923,E2 331.483} C_DIS
LIN {X -38.5912,Y 80.8037,Z 89,A 109.4375,B 24.9075,C -2.2203,E1 24.9333,E2 335.5957} C_DIS
LIN {X -34.3498,Y 82.6969,Z 89,A 106.9387,B 24.906,C -2.239,E1 24.9396,E2 338.0559} C_DIS
LIN {X -30.6768,Y 84.1273,Z 89,A 103.3554,B 24.9084,C -2.21,E1 24.9492,E2 341.7156} C_DIS
LIN {X -26.3973,Y 85.5668,Z 89,A 101.5401,B 24.9054,C -2.2462,E1 24.9538,E2 343.4481} C_DIS
LIN {X -23.9887,Y 86.274,Z 89,A 99.2295,B 24.907,C -2.2262,E1 24.9601,E2 345.81} C_DIS
LIN {X -20.8745,Y 87.0796,Z 89,A 97.3973,B 24.9063,C -2.2351,E1 24.965,E2 347.6236} C_DIS
LIN {X -16.2645,Y 88.0574,Z 89,A 94.6842,B 24.9053,C -2.2469,E1 24.9724,E2 350.3116} C_DIS
LIN {X -13.5099,Y 88.5211,Z 89,A 92.9253,B 24.9051,C -2.2491,E1 24.9772,E2 352.067} C_DIS
LIN {X -10.7118,Y 88.9034,Z 89,A 90.7753,B 24.9059,C -2.2394,E1 24.9833,E2 354.2415} C_DIS
LIN {X -7.5484,Y 89.2282,Z 89,A 88.8321,B 24.9056,C -2.2432,E1 24.9886,E2 356.1765} C_DIS
LIN {X -3.9339,Y 89.4595,Z 89,A 86.7644,B 24.9049,C -2.252,E1 24.9943,E2 358.224} C_DIS
LIN {X -1.1692,Y 89.5396,Z 89,A 84.912,B 24.905,C -2.2498,E1 24.9995,E2 360.0818} C_DIS
LIN {X 1.9385,Y 89.5254,Z 89,A 82.8546,B 24.9052,C -2.2479,E1 25.0053,E2 362.1434} C_DIS
LIN {X 5.3303,Y 89.388,Z 89,A 80.9661,B 24.9044,C -2.2571,E1 25.0105,E2 364.0096} C_DIS
LIN {X 9.0152,Y 89.0915,Z 89,A 78.3816,B 24.905,C -2.2498,E1 25.0177,E2 366.6098} C_DIS
LIN {X 12.1074,Y 88.7245,Z 89,A 76.3069,B 24.9053,C -2.2468,E1 25.0235,E2 368.6901} C_DIS
LIN {X 15.2287,Y 88.2427,Z 89,A 73.8772,B 24.9065,C -2.2329,E1 25.0303,E2 371.1502} C_DIS
LIN {X 18.4116,Y 87.6336,Z 89,A 72.471,B 24.9047,C -2.2536,E1 25.034,E2 372.5057} C_DIS
LIN {X 20.9431,Y 87.0628,Z 89,A 70.6012,B 24.9054,C -2.2459,E1 25.0391,E2 374.391} C_DIS
LIN {X 24.262,Y 86.1966,Z 89,A 68.4142,B 24.9054,C -2.2447,E1 25.045,E2 376.5774} C_DIS
LIN {X 28.3474,Y 84.941,Z 89,A 65.9328,B 24.905,C -2.2509,E1 25.0516,E2 379.0395} C_DIS
LIN {X 31.2466,Y 83.9177,Z 89,A 62.6435,B 24.9087,C -2.2058,E1 25.0604,E2 382.4287} C_DIS
LIN {X 36.2217,Y 81.8944,Z 89,A 60.4769,B 24.9056,C -2.2438,E1 25.0657,E2 384.5001} C_DIS
LIN {X 38.7022,Y 80.7503,Z 89,A 58.6779,B 24.9059,C -2.2401,E1 25.0703,E2 386.3034} C_DIS
LIN {X 43.9159,Y 78.0382,Z 89,A 55.4207,B 24.9049,C -2.252,E1 25.0783,E2 389.5231} C_DIS
LIN {X 47.3879,Y 75.9793,Z 89,A 51.7477,B 24.9083,C -2.2115,E1 25.0873,E2 393.2807} C_DIS
LIN {X 50.1705,Y 74.1714,Z 89,A 50.5904,B 24.9058,C -2.2407,E1 25.0898,E2 394.365} C_DIS
LIN {X 53.1868,Y 72.04,Z 89,A 47.0263,B 24.9095,C -2.196,E1 25.0981,E2 398.0223} C_DIS
LIN {X 56.4587,Y 69.5046,Z 89,A 45.1751,B 24.9077,C -2.2181,E1 25.102,E2 399.8143} C_DIS
LIN {X 61.3552,Y 65.2228,Z 89,A 41.1431,B 24.908,C -2.2143,E1 25.1104,E2 403.8393} C_DIS
LIN {X 63.416,Y 63.2223,Z 89,A 39.0575,B 24.9091,C -2.2019,E1 25.1145,E2 405.9453} C_DIS
LIN {X 67.6224,Y 58.7005,Z 89,A 35.428,B 24.9089,C -2.2042,E1 25.1214,E2 409.5534} C_DIS
LIN {X 69.3502,Y 56.6493,Z 89,A 32.4533,B 24.9127,C -2.157,E1 25.1268,E2 412.6259} C_DIS
LIN {X 72.5745,Y 52.4568,Z 89,A 30.3163,B 24.9099,C -2.1916,E1 25.1302,E2 414.671} C_DIS
LIN {X 74.655,Y 49.4483,Z 89,A 26.9393,B 24.9133,C -2.1498,E1 25.1355,E2 418.13} C_DIS
LIN {X 77.1167,Y 45.5136,Z 89,A 23.685,B 24.9147,C -2.1321,E1 25.1402,E2 421.4091} C_DIS
LIN {X 79.8458,Y 40.5362,Z 89,A 21.8912,B 24.9103,C -2.1863,E1 25.1423,E2 423.0656} C_DIS
LIN {X 81.6415,Y 36.785,Z 89,A 18.7007,B 24.9125,C -2.1601,E1 25.1462,E2 426.3008} C_DIS
LIN {X 83.6148,Y 32.0494,Z 89,A 15.6316,B 24.9126,C -2.1581,E1 25.1495,E2 429.3576} C_DIS
LIN {X 84.7325,Y 28.9658,Z 89,A 12.7372,B 24.9154,C -2.1239,E1 25.1522,E2 432.3165} C_DIS
LIN {X 85.7791,Y 25.6999,Z 89,A 10.6239,B 24.9157,C -2.1201,E1 25.1539,E2 434.4267} C_DIS
LIN {X 86.6522,Y 22.5824,Z 89,A 9.341,B 24.914,C -2.1417,E1 25.1548,E2 435.6512} C_DIS
LIN {X 87.4756,Y 19.144,Z 89,A 6.3308,B 24.9166,C -2.1083,E1 25.1567,E2 438.7229} C_DIS
LIN {X 88.2061,Y 15.4381,Z 89,A 4.1903,B 24.9165,C -2.1105,E1 25.1577,E2 440.8457} C_DIS
LIN {X 88.8018,Y 11.5203,Z 89,A 1.9239,B 24.9163,C -2.1121,E1 25.1586,E2 443.0949} C_DIS
LIN {X 89.1572,Y 8.3358,Z 89,A -0.1304,B 24.9169,C -2.1055,E1 25.1592,E2 445.1527} C_DIS
LIN {X 89.4053,Y 5.0161,Z 89,A -2.2231,B 24.9173,C -2.1,E1 25.1596,E2 447.2458} C_DIS
LIN {X 89.5004,Y 2.8562,Z 89,A -3.6368,B 24.9177,C -2.0945,E1 25.1597,E2 448.6641} C_DIS
LIN {X 89.5434,Y -0.7641,Z 89,A -5.8806,B 24.9181,C -2.0897,E1 25.1597,E2 450.906} C_DIS
LIN {X 89.4602,Y -3.9183,Z 89,A -8.0526,B 24.919,C -2.0778,E1 25.1595,E2 453.0931} C_DIS
LIN {X 89.227,Y -7.5633,Z 89,A -10.3176,B 24.9194,C -2.0728,E1 25.1591,E2 455.3565} C_DIS
LIN {X 88.7526,Y -11.8998,Z 89,A -13.2734,B 24.9206,C -2.058,E1 25.1581,E2 458.3297} C_DIS
LIN {X 88.039,Y -16.3673,Z 89,A -15.9688,B 24.9207,C -2.0559,E1 25.1568,E2 461.0144} C_DIS
LIN {X 87.1722,Y -20.4841,Z 89,A -18.4468,B 24.9208,C -2.055,E1 25.1554,E2 463.4801} C_DIS
LIN {X 86.524,Y -23.0686,Z 89,A -20.3139,B 24.9217,C -2.0438,E1 25.154,E2 465.3627} C_DIS
LIN {X 85.6212,Y -26.2218,Z 89,A -22.4006,B 24.9221,C -2.0376,E1 25.1524,E2 467.4521} C_DIS
LIN {X 83.8535,Y -31.4191,Z 89,A -25.7035,B 24.9224,C -2.0342,E1 25.1494,E2 470.7444} C_DIS
LIN {X 81.7345,Y -36.5787,Z 89,A -29.0675,B 24.9227,C -2.0307,E1 25.1458,E2 474.0984} C_DIS
LIN {X 80.2259,Y -39.7779,Z 89,A -31.678,B 24.9241,C -2.0115,E1 25.1426,E2 476.74} C_DIS
LIN {X 78.5672,Y -42.9622,Z 89,A -34.1429,B 24.9251,C -1.9988,E1 25.1393,E2 479.2219} C_DIS
LIN {X 76.7053,Y -46.2048,Z 89,A -36.0811,B 24.9244,C -2.0081,E1 25.1366,E2 481.1283} C_DIS
LIN {X 73.9113,Y -50.5547,Z 89,A -39.3962,B 24.9251,C -1.9985,E1 25.1316,E2 484.4494} C_DIS
LIN {X 71.6559,Y -53.7021,Z 89,A -41.982,B 24.9259,C -1.9879,E1 25.1273,E2 487.0477} C_DIS
LIN {X 69.9916,Y -55.8553,Z 89,A -43.8035,B 24.9265,C -1.9804,E1 25.1242,E2 488.8783} C_DIS
LIN {X 67.1957,Y -59.1891,Z 89,A -46.9493,B 24.9279,C -1.9606,E1 25.1184,E2 492.0568} C_DIS
LIN {X 63.2322,Y -63.4062,Z 89,A -50.6682,B 24.9286,C -1.9509,E1 25.1111,E2 495.7824} C_DIS
LIN {X 59.429,Y -66.9837,Z 89,A -54.0417,B 24.9293,C -1.9421,E1 25.1041,E2 499.1634} C_DIS
LIN {X 53.8612,Y -71.5363,Z 89,A -57.7363,B 24.9277,C -1.9636,E1 25.0963,E2 502.7932} C_DIS
LIN {X 51.0079,Y -73.5981,Z 89,A -60.302,B 24.9289,C -1.948,E1 25.0904,E2 505.3867} C_DIS
LIN {X 46.3954,Y -76.5895,Z 89,A -63.8189,B 24.9293,C -1.9413,E1 25.0821,E2 508.9081} C_DIS
LIN {X 41.385,Y -79.4097,Z 89,A -67.3924,B 24.9296,C -1.9384,E1 25.0734,E2 512.4779} C_DIS
LIN {X 39.0051,Y -80.6048,Z 89,A -69.2884,B 24.9302,C -1.9291,E1 25.0686,E2 514.3909} C_DIS
LIN {X 35.8483,Y -82.0572,Z 89,A -72.0642,B 24.9318,C -1.907,E1 25.0614,E2 517.2122} C_DIS
LIN {X 32.5221,Y -83.4316,Z 89,A -73.556,B 24.9301,C -1.9312,E1 25.0576,E2 518.6433} C_DIS
LIN {X 27.8151,Y -85.1167,Z 89,A -76.7109,B 24.9303,C -1.9286,E1 25.0494,E2 521.798} C_DIS
LIN {X 23.3094,Y -86.4589,Z 89,A -79.4629,B 24.9299,C -1.9339,E1 25.042,E2 524.5328} C_DIS
LIN {X 21.1441,Y -87.0138,Z 89,A -81.289,B 24.931,C -1.919,E1 25.037,E2 526.3912} C_DIS
LIN {X 18.1102,Y -87.6955,Z 89,A -84.2035,B 24.9333,C -1.8866,E1 25.0288,E2 529.379} C_DIS
LIN {X 13.7919,Y -88.4775,Z 89,A -85.7711,B 24.9305,C -1.9256,E1 25.0248,E2 530.8526} C_DIS
LIN {X 10.1722,Y -88.9666,Z 89,A -88.5232,B 24.9316,C -1.9102,E1 25.017,E2 533.6388} C_DIS
LIN {X 6.7668,Y -89.2906,Z 89,A -90.7016,B 24.9316,C -1.9095,E1 25.011,E2 535.8178} C_DIS
LIN {X 3.1589,Y -89.4907,Z 89,A -93.7156,B 24.9333,C -1.8857,E1 25.0024,E2 538.8873} C_DIS
LIN {X 3.1589,Y -89.4907,Z 89,A -93.7156,B 24.9333,C -1.8857,E1 25.0024,E2 538.8873} C_DIS
Enddeposition()
LIN {X 0.5766,Y -88.5355,Z 89,A -94.0926,B 24.9291,C -1.9445,E1 25.0018,E2 539.1248} C_DIS
Startdeposition()
$VEL.CP = VEL_PRINT
LIN {X 4.7576,Y -88.4249,Z 89,A -91.1296,B 24.9284,C -1.9536,E1 25.0101,E2 536.1409} C_DIS
LIN {X 7.5576,Y -88.231,Z 89,A -89.1019,B 24.9279,C -1.9615,E1 25.0158,E2 534.0956} C_DIS
LIN {X 11.123,Y -87.8517,Z 89,A -86.857,B 24.9279,C -1.9604,E1 25.022,E2 531.8549} C_DIS
LIN {X 15.4058,Y -87.2027,Z 89,A -83.7622,B 24.9271,C -1.9723,E1 25.0306,E2 528.735} C_DIS
LIN {X 19.9261,Y -86.2817,Z 89,A -81.279,B 24.9281,C -1.9581,E1 25.0373,E2 526.2888} C_DIS
LIN {X 22.5549,Y -85.6337,Z 89,A -78.9596,B 24.9266,C -1.9791,E1 25.0437,E2 523.9233} C_DIS
LIN {X 27.0789,Y -84.311,Z 89,A -76.5956,B 24.928,C -1.9593,E1 25.0498,E2 521.6102} C_DIS
LIN {X 31.4703,Y -82.772,Z 89,A -73.4478,B 24.9274,C -1.9678,E1 25.0582,E2 518.4486} C_DIS
LIN {X 35.5575,Y -81.1004,Z 89,A -70.2436,B 24.9262,C -1.9839,E1 25.0665,E2 515.2141} C_DIS
LIN {X 38.9477,Y -79.5289,Z 89,A -68.0387,B 24.9265,C -1.9804,E1 25.072,E2 513.0232} C_DIS
LIN {X 42.5057,Y -77.6845,Z 89,A -65.0084,B 24.925,C -2,E1 25.0795,E2 509.9552} C_DIS
LIN {X 45.321,Y -76.0768,Z 89,A -63.4123,B 24.926,C -1.9864,E1 25.0833,E2 508.3962} C_DIS
LIN {X 49.3272,Y -73.5429,Z 89,A -60.4928,B 24.926,C -1.9871,E1 25.0901,E2 505.4843} C_DIS
LIN {X 53.8186,Y -70.3223,Z 89,A -56.7821,B 24.9251,C -1.9992,E1 25.0985,E2 501.7583} C_DIS
LIN {X 58.6618,Y -66.3376,Z 89,A -52.1038,B 24.9227,C -2.0301,E1 25.1086,E2 497.025} C_DIS
LIN {X 61.3736,Y -63.8348,Z 89,A -50.4044,B 24.9241,C -2.0115,E1 25.1119,E2 495.3766} C_DIS
LIN {X 63.6126,Y -61.6037,Z 89,A -47.5972,B 24.9217,C -2.0435,E1 25.1175,E2 492.5059} C_DIS
LIN {X 66.4196,Y -58.5679,Z 89,A -44.7982,B 24.9208,C -2.0547,E1 25.1227,E2 489.6929} C_DIS
LIN {X 69.3266,Y -55.095,Z 89,A -42.918,B 24.9231,C -2.025,E1 25.1259,E2 487.8916} C_DIS
LIN {X 72.7275,Y -50.5202,Z 89,A -39.594,B 24.9233,C -2.0221,E1 25.1314,E2 484.5904} C_DIS
LIN {X 75.0244,Y -47.0419,Z 89,A -36.4126,B 24.9214,C -2.0468,E1 25.1363,E2 481.3666} C_DIS
LIN {X 77.8574,Y -42.1877,Z 89,A -32.7821,B 24.9206,C -2.0571,E1 25.1413,E2 477.7307} C_DIS
LIN {X 79.46,Y -39.0866,Z 89,A -30.1649,B 24.9191,C -2.0766,E1 25.1446,E2 475.0814} C_DIS
LIN {X 81.8587,Y -33.7756,Z 89,A -26.8337,B 24.9195,C -2.0722,E1 25.1483,E2 471.7786} C_DIS
LIN {X 83.0004,Y -30.8675,Z 89,A -24.8269,B 24.919,C -2.0779,E1 25.1503,E2 469.7697} C_DIS
LIN {X 84.9099,Y -25.1375,Z 89,A -20.9256,B 24.9181,C -2.0898,E1 25.1537,E2 465.8624} C_DIS
LIN {X 85.8047,Y -21.8896,Z 89,A -18.0423,B 24.9155,C -2.1221,E1 25.1557,E2 462.9196} C_DIS
LIN {X 86.7071,Y -17.9859,Z 89,A -16.007,B 24.9165,C -2.1102,E1 25.1569,E2 460.9243} C_DIS
LIN {X 87.4249,Y -14.0971,Z 89,A -13.5096,B 24.916,C -2.1161,E1 25.158,E2 458.4275} C_DIS
LIN {X 87.9584,Y -10.2424,Z 89,A -11.242,B 24.916,C -2.1152,E1 25.1588,E2 456.1753} C_DIS
LIN {X 88.3415,Y -6.1134,Z 89,A -8.1496,B 24.9142,C -2.1385,E1 25.1596,E2 453.0462} C_DIS
LIN {X 88.5482,Y -1.0233,Z 89,A -5.1508,B 24.9142,C -2.1384,E1 25.1598,E2 450.0656} C_DIS
LIN {X 88.5179,Y 2.4908,Z 89,A -2.7232,B 24.9132,C -2.1512,E1 25.1596,E2 447.6222} C_DIS
LIN {X 88.2791,Y 6.9566,Z 89,A -0.388,B 24.9141,C -2.1404,E1 25.1593,E2 445.3264} C_DIS
LIN {X 88.0405,Y 9.5148,Z 89,A 1.4866,B 24.913,C -2.1532,E1 25.1587,E2 443.4327} C_DIS
LIN {X 87.6184,Y 12.8349,Z 89,A 4.1129,B 24.9111,C -2.1765,E1 25.1577,E2 440.7668} C_DIS
LIN {X 86.1854,Y 20.343,Z 89,A 8.4939,B 24.9115,C -2.1716,E1 25.1553,E2 436.423} C_DIS
LIN {X 85.119,Y 24.4216,Z 89,A 11.4281,B 24.9103,C -2.1872,E1 25.1531,E2 433.4688} C_DIS
LIN {X 83.3691,Y 29.8569,Z 89,A 15.1031,B 24.9094,C -2.1974,E1 25.1499,E2 429.7903} C_DIS
LIN {X 81.858,Y 33.7791,Z 89,A 17.5792,B 24.9094,C -2.1967,E1 25.1474,E2 427.3297} C_DIS
LIN {X 80.6908,Y 36.4772,Z 89,A 19.6344,B 24.9086,C -2.2075,E1 25.145,E2 425.2601} C_DIS
LIN {X 78.9794,Y 40.0489,Z 89,A 22.9667,B 24.9057,C -2.2419,E1 25.1408,E2 421.8643} C_DIS
LIN {X 76.9422,Y 43.8358,Z 89,A 24.7594,B 24.908,C -2.2144,E1 25.1384,E2 420.146} C_DIS
LIN {X 75.896,Y 45.6241,Z 89,A 26.5189,B 24.9065,C -2.2327,E1 25.1359,E2 418.3524} C_DIS
LIN {X 73.572,Y 49.2843,Z 89,A 29.1063,B 24.9065,C -2.2322,E1 25.1319,E2 415.779} C_DIS
LIN {X 71.7695,Y 51.875,Z 89,A 31.3757,B 24.9054,C -2.2452,E1 25.1282,E2 413.4898} C_DIS
LIN {X 68.7976,Y 55.7536,Z 89,A 34.3471,B 24.9054,C -2.2462,E1 25.1231,E2 410.5302} C_DIS
LIN {X 66.4761,Y 58.5028,Z 89,A 37.4652,B 24.9026,C -2.2791,E1 25.1173,E2 407.3483} C_DIS
LIN {X 63.279,Y 61.9477,Z 89,A 39.4044,B 24.9053,C -2.2473,E1 25.1137,E2 405.4926} C_DIS
LIN {X 61.2209,Y 63.9819,Z 89,A 42.5181,B 24.9012,C -2.2943,E1 25.1072,E2 402.2807} C_DIS
LIN {X 57.3647,Y 67.4597,Z 89,A 44.6646,B 24.9043,C -2.2588,E1 25.1028,E2 400.2265} C_DIS
LIN {X 54.7318,Y 69.6137,Z 89,A 47.445,B 24.9022,C -2.2827,E1 25.0967,E2 397.4001} C_DIS
LIN {X 51.7405,Y 71.8655,Z 89,A 49.3986,B 24.9033,C -2.2708,E1 25.0923,E2 395.4815} C_DIS
LIN {X 49.3638,Y 73.5181,Z 89,A 51.5419,B 24.9022,C -2.2831,E1 25.0873,E2 393.3164} C_DIS
LIN {X 44.5428,Y 76.536,Z 89,A 54.774,B 24.903,C -2.2734,E1 25.0797,E2 390.1174} C_DIS
LIN {X 42.1818,Y 77.8606,Z 89,A 57.1384,B 24.9011,C -2.2964,E1 25.0738,E2 387.7051} C_DIS
LIN {X 38.9272,Y 79.539,Z 89,A 59.318,B 24.9014,C -2.2929,E1 25.0684,E2 385.5397} C_DIS
LIN {X 35.6662,Y 81.053,Z 89,A 61.592,B 24.9013,C -2.2938,E1 25.0626,E2 383.2693} C_DIS
LIN {X 30.1202,Y 83.2731,Z 89,A 65.1979,B 24.9017,C -2.2889,E1 25.0533,E2 379.6829} C_DIS
LIN {X 27.1265,Y 84.2956,Z 89,A 67.5083,B 24.9008,C -2.2993,E1 25.0471,E2 377.3522} C_DIS
LIN {X 23.9093,Y 85.2642,Z 89,A 69.9686,B 24.8999,C -2.3102,E1 25.0404,E2 374.8701} C_DIS
LIN {X 20.5623,Y 86.1334,Z 89,A 71.5072,B 24.9017,C -2.2885,E1 25.0364,E2 373.3853} C_DIS
LIN {X 14.643,Y 87.3336,Z 89,A 75.2858,B 24.902,C -2.2859,E1 25.0261,E2 369.6173} C_DIS
LIN {X 10.9731,Y 87.8711,Z 89,A 77.7136,B 24.9018,C -2.2874,E1 25.0193,E2 367.1881} C_DIS
LIN {X 7.5143,Y 88.2345,Z 89,A 80.2892,B 24.9009,C -2.2981,E1 25.0121,E2 364.5887} C_DIS
LIN {X 3.322,Y 88.4917,Z 89,A 83.2835,B 24.9001,C -2.3069,E1 25.0037,E2 361.5744} C_DIS
LIN {X -1.4605,Y 88.5408,Z 89,A 86.0212,B 24.9012,C -2.2949,E1 24.9961,E2 358.8655} C_DIS
LIN {X -4.7036,Y 88.4279,Z 89,A 88.6268,B 24.8999,C -2.3103,E1 24.9888,E2 356.2226} C_DIS
LIN {X -7.9576,Y 88.1946,Z 89,A 89.8679,B 24.9023,C -2.2817,E1 24.9855,E2 355.0488} C_DIS
LIN {X -11.5602,Y 87.7951,Z 89,A 92.4486,B 24.9018,C -2.2878,E1 24.9783,E2 352.452} C_DIS
LIN {X -14.4437,Y 87.367,Z 89,A 94.4404,B 24.9016,C -2.2898,E1 24.9728,E2 350.4536} C_DIS
LIN {X -19.3245,Y 86.4191,Z 89,A 97.6167,B 24.902,C -2.2859,E1 24.9641,E2 347.2831} C_DIS
LIN {X -23.6532,Y 85.3355,Z 89,A 100.5713,B 24.902,C -2.2851,E1 24.9561,E2 344.326} C_DIS
LIN {X -26.1064,Y 84.6171,Z 89,A 103.0588,B 24.9,C -2.3092,E1 24.9493,E2 341.7767} C_DIS
LIN {X -30.1654,Y 83.2566,Z 89,A 105.2776,B 24.9017,C -2.2885,E1 24.9436,E2 339.6027} C_DIS
LIN {X -34.0589,Y 81.7417,Z 89,A 108.2258,B 24.9014,C -2.2923,E1 24.9359,E2 336.6388} C_DIS
LIN {X -38.3443,Y 79.8204,Z 89,A 111.0247,B 24.9024,C -2.2803,E1 24.9289,E2 333.8616} C_DIS
LIN {X -42.0935,Y 77.9085,Z 89,A 113.5487,B 24.9034,C -2.2697,E1 24.9227,E2 331.3559} C_DIS
LIN {X -46.6905,Y 75.2439,Z 89,A 117.5673,B 24.9024,C -2.2812,E1 24.913,E2 327.2977} C_DIS
LIN {X -49.6588,Y 73.3184,Z 89,A 119.1979,B 24.9045,C -2.2568,E1 24.9093,E2 325.7198} C_DIS
LIN {X -52.6871,Y 71.1733,Z 89,A 122.2898,B 24.9031,C -2.2727,E1 24.9023,E2 322.5791} C_DIS
LIN {X -55.5485,Y 68.9638,Z 89,A 124.3646,B 24.9042,C -2.2597,E1 24.8978,E2 320.5276} C_DIS
LIN {X -58.4894,Y 66.4881,Z 89,A 126.5207,B 24.9055,C -2.2442,E1 24.8933,E2 318.3999} C_DIS
LIN {X -61.8295,Y 63.3933,Z 89,A 129.7153,B 24.9055,C -2.2447,E1 24.8868,E2 315.191} C_DIS
LIN {X -65.2256,Y 59.8933,Z 89,A 132.6185,B 24.9068,C -2.2295,E1 24.8812,E2 312.3115} C_DIS
LIN {X -67.1152,Y 57.7697,Z 89,A 134.7798,B 24.9064,C -2.2343,E1 24.8772,E2 310.1289} C_DIS
LIN {X -69.6699,Y 54.6605,Z 89,A 137.0842,B 24.9077,C -2.2187,E1 24.8733,E2 307.851} C_DIS
LIN {X -71.8425,Y 51.7705,Z 89,A 139.8654,B 24.9071,C -2.2254,E1 24.8686,E2 305.0404} C_DIS
LIN {X -74.5251,Y 47.8288,Z 89,A 142.7847,B 24.9082,C -2.2119,E1 24.8642,E2 302.1386} C_DIS
LIN {X -76.6937,Y 44.2684,Z 89,A 145.9208,B 24.9078,C -2.2171,E1 24.8597,E2 298.9738} C_DIS
LIN {X -78.433,Y 41.1081,Z 89,A 147.4258,B 24.9104,C -2.186,E1 24.8578,E2 297.535} C_DIS
LIN {X -79.5083,Y 38.9892,Z 89,A 149.4476,B 24.9096,C -2.1956,E1 24.8553,E2 295.4795} C_DIS
LIN {X -81.2,Y 35.329,Z 89,A 151.8469,B 24.9107,C -2.1817,E1 24.8525,E2 293.1002} C_DIS
LIN {X -82.4532,Y 32.2965,Z 89,A 154.78,B 24.9093,C -2.1989,E1 24.8495,E2 290.1095} C_DIS
LIN {X -83.9111,Y 28.2934,Z 89,A 156.5276,B 24.9124,C -2.1609,E1 24.848,E2 288.4427} C_DIS
LIN {X -85.283,Y 23.8431,Z 89,A 159.3461,B 24.9136,C -2.1459,E1 24.8457,E2 285.6438} C_DIS
LIN {X -86.4882,Y 19.0101,Z 89,A 163.1968,B 24.913,C -2.1539,E1 24.8431,E2 281.7515} C_DIS
LIN {X -87.0993,Y 15.9811,Z 89,A 164.9737,B 24.914,C -2.141,E1 24.8422,E2 279.9948} C_DIS
LIN {X -87.584,Y 13.0708,Z 89,A 167.967,B 24.912,C -2.1666,E1 24.841,E2 276.9226} C_DIS
LIN {X -88.1683,Y 8.2424,Z 89,A 169.7149,B 24.916,C -2.1158,E1 24.8405,E2 275.2856} C_DIS
LIN {X -88.5155,Y 2.5701,Z 89,A 173.641,B 24.9164,C -2.1111,E1 24.8398,E2 271.347} C_DIS
LIN {X -88.5485,Y -0.9092,Z 89,A 176.2145,B 24.9162,C -2.1132,E1 24.8398,E2 268.7529} C_DIS
LIN {X -88.3214,Y -6.4114,Z 89,A 179.5049,B 24.9178,C -2.0939,E1 24.8403,E2 265.4888} C_DIS
LIN {X -88.1095,Y -8.8562,Z 89,A -178.0017,B 24.9161,C -2.1154,E1 24.841,E2 262.9293} C_DIS
LIN {X -87.6325,Y -12.7361,Z 89,A -176.2953,B 24.9186,C -2.0834,E1 24.8416,E2 261.2891} C_DIS
LIN {X -86.6654,Y -18.189,Z 89,A -172.7575,B 24.9196,C -2.0709,E1 24.8434,E2 257.7602} C_DIS
LIN {X -86.1211,Y -20.6127,Z 89,A -170.5775,B 24.9187,C -2.0827,E1 24.8448,E2 255.5391} C_DIS
LIN {X -85.1698,Y -24.2425,Z 89,A -168.5487,B 24.9201,C -2.0636,E1 24.8463,E2 253.544} C_DIS
LIN {X -84.1968,Y -27.4318,Z 89,A -166.2656,B 24.9204,C -2.0609,E1 24.8482,E2 251.2544} C_DIS
LIN {X -82.9897,Y -30.8957,Z 89,A -164.016,B 24.9212,C -2.0503,E1 24.8503,E2 249.0175} C_DIS
LIN {X -81.8977,Y -33.6816,Z 89,A -161.9052,B 24.9212,C -2.0498,E1 24.8525,E2 246.8958} C_DIS
LIN {X -79.7903,Y -38.407,Z 89,A -159.1285,B 24.9232,C -2.0236,E1 24.8557,E2 244.1665} C_DIS
LIN {X -77.9499,Y -42.0171,Z 89,A -156.016,B 24.9227,C -2.0308,E1 24.8597,E2 241.0202} C_DIS
LIN {X -76.6008,Y -44.4301,Z 89,A -154.0787,B 24.9227,C -2.0304,E1 24.8624,E2 239.0736} C_DIS
LIN {X -74.7293,Y -47.5106,Z 89,A -151.7507,B 24.9232,C -2.0242,E1 24.8658,E2 236.7485} C_DIS
LIN {X -71.8606,Y -51.7473,Z 89,A -148.4531,B 24.9238,C -2.0156,E1 24.8711,E2 233.4553} C_DIS
LIN {X -69.1459,Y -55.3237,Z 89,A -145.6708,B 24.9246,C -2.0049,E1 24.8758,E2 230.6853} C_DIS
LIN {X -66.0871,Y -58.9415,Z 89,A -142.0708,B 24.9239,C -2.0141,E1 24.8825,E2 227.0471} C_DIS
LIN {X -61.5521,Y -63.6627,Z 89,A -137.7542,B 24.9244,C -2.0076,E1 24.891,E2 222.7276} C_DIS
LIN {X -59.2082,Y -65.8483,Z 89,A -136.282,B 24.9261,C -1.9851,E1 24.8939,E2 221.303} C_DIS
LIN {X -57.0744,Y -67.7075,Z 89,A -134.136,B 24.9257,C -1.9912,E1 24.8985,E2 219.1341} C_DIS
LIN {X -54.5745,Y -69.7379,Z 89,A -132.4085,B 24.9268,C -1.9765,E1 24.9022,E2 217.4353} C_DIS
LIN {X -52.5828,Y -71.2512,Z 89,A -130.3899,B 24.926,C -1.986,E1 24.9068,E2 215.3868} C_DIS
LIN {X -47.7948,Y -74.5469,Z 89,A -127.2705,B 24.928,C -1.9602,E1 24.9139,E2 212.3185} C_DIS
LIN {X -45.8189,Y -75.7776,Z 89,A -125.2078,B 24.9269,C -1.9752,E1 24.9189,E2 210.2137} C_DIS
LIN {X -42.6284,Y -77.6184,Z 89,A -123.1247,B 24.9278,C -1.9625,E1 24.9239,E2 208.1546} C_DIS
LIN {X -39.6004,Y -79.2053,Z 89,A -120.7666,B 24.9277,C -1.9643,E1 24.9298,E2 205.7859} C_DIS
LIN {X -36.5716,Y -80.6483,Z 89,A -117.9633,B 24.9264,C -1.9818,E1 24.937,E2 202.934} C_DIS
LIN {X -33.3937,Y -82.0149,Z 89,A -116.6653,B 24.9287,C -1.9498,E1 24.9402,E2 201.7091} C_DIS
LIN {X -31.2476,Y -82.8564,Z 89,A -114.8277,B 24.928,C -1.9593,E1 24.945,E2 199.845} C_DIS
LIN {X -26.9682,Y -84.3468,Z 89,A -111.6399,B 24.9276,C -1.9651,E1 24.9535,E2 196.6376} C_DIS
LIN {X -23.7815,Y -85.3004,Z 89,A -109.6297,B 24.928,C -1.9591,E1 24.9589,E2 194.6383} C_DIS
LIN {X -17.5596,Y -86.7946,Z 89,A -105.7031,B 24.9287,C -1.9502,E1 24.9695,E2 190.7278} C_DIS
LIN {X -13.9543,Y -87.4474,Z 89,A -103.2812,B 24.9287,C -1.951,E1 24.9762,E2 188.3015} C_DIS
LIN {X -11.268,Y -87.8329,Z 89,A -101.3676,B 24.9283,C -1.9558,E1 24.9815,E2 186.3751} C_DIS
LIN {X -7.7204,Y -88.2165,Z 89,A -98.6355,B 24.9273,C -1.9695,E1 24.9892,E2 183.609} C_DIS
LIN {X -3.7947,Y -88.4714,Z 89,A -96.6728,B 24.9287,C -1.9505,E1 24.9946,E2 181.6908} C_DIS
LIN {X -0.9111,Y -88.5488,Z 89,A -94.1584,B 24.9271,C -1.9722,E1 25.0018,E2 179.1248} C_DIS
LIN {X -0.9111,Y -88.5488,Z 89,A -94.1584,B 24.9271,C -1.9722,E1 25.0018,E2 179.1248} C_DIS
Enddeposition()
LIN {X 0.5712,Y -87.548,Z 89,A -94.3147,B 24.9285,C -1.9533,E1 25.0012,E2 179.3261} C_DIS
Startdeposition()
$VEL.CP = VEL_PRINT
LIN {X -2.7189,Y -87.5173,Z 89,A -96.5352,B 24.9287,C -1.9505,E1 24.995,E2 181.5532} C_DIS
LIN {X -6.5587,Y -87.3145,Z 89,A -99.4513,B 24.9296,C -1.9377,E1 24.9868,E2 184.5008} C_DIS
LIN {X -10.0328,Y -86.9829,Z 89,A -101.6605,B 24.9294,C -1.9403,E1 24.9806,E2 186.7051} C_DIS
LIN {X -13.0079,Y -86.5887,Z 89,A -104.3044,B 24.9309,C -1.9195,E1 24.9732,E2 189.4006} C_DIS
LIN {X -16.6322,Y -85.9653,Z 89,A -105.5335,B 24.9282,C -1.9571,E1 24.9701,E2 190.5415} C_DIS
LIN {X -20.7575,Y -85.0634,Z 89,A -108.8407,B 24.9293,C -1.9413,E1 24.9609,E2 193.8904} C_DIS
LIN {X -26.1215,Y -83.5725,Z 89,A -112.673,B 24.9296,C -1.9379,E1 24.9506,E2 197.737} C_DIS
LIN {X -29.623,Y -82.3972,Z 89,A -114.9094,B 24.929,C -1.9455,E1 24.9447,E2 199.9598} C_DIS
LIN {X -32.4581,Y -81.3226,Z 89,A -116.9022,B 24.929,C -1.9471,E1 24.9396,E2 201.9531} C_DIS
LIN {X -37.427,Y -79.1591,Z 89,A -120.4602,B 24.9287,C -1.9506,E1 24.9305,E2 205.5113} C_DIS
LIN {X -39.8076,Y -77.9873,Z 89,A -122.2859,B 24.9287,C -1.9501,E1 24.9259,E2 207.3431} C_DIS
LIN {X -42.451,Y -76.581,Z 89,A -124.2279,B 24.9285,C -1.9532,E1 24.9212,E2 209.2832} C_DIS
LIN {X -45.3698,Y -74.8883,Z 89,A -126.3225,B 24.928,C -1.9598,E1 24.9161,E2 211.3685} C_DIS
LIN {X -48.1821,Y -73.1105,Z 89,A -129.389,B 24.9297,C -1.9367,E1 24.9088,E2 214.4999} C_DIS
LIN {X -51.736,Y -70.6403,Z 89,A -131.3278,B 24.9274,C -1.9679,E1 24.9046,E2 216.3711} C_DIS
LIN {X -54.2847,Y -68.701,Z 89,A -133.4362,B 24.9271,C -1.9713,E1 24.8999,E2 218.4793} C_DIS
LIN {X -56.6737,Y -66.7441,Z 89,A -135.5177,B 24.927,C -1.9732,E1 24.8955,E2 220.5641} C_DIS
LIN {X -58.9858,Y -64.7103,Z 89,A -138.6409,B 24.9291,C -1.9449,E1 24.8889,E2 223.7673} C_DIS
LIN {X -62.7074,Y -61.112,Z 89,A -141.0259,B 24.9264,C -1.9811,E1 24.8843,E2 226.0762} C_DIS
LIN {X -67.1399,Y -56.2049,Z 89,A -145.3073,B 24.9256,C -1.9922,E1 24.8764,E2 230.3505} C_DIS
LIN {X -70.5643,Y -51.8397,Z 89,A -148.665,B 24.9243,C -2.0088,E1 24.8707,E2 233.6845} C_DIS
LIN {X -73.0065,Y -48.3398,Z 89,A -151.7713,B 24.9245,C -2.0067,E1 24.8658,E2 236.8112} C_DIS
LIN {X -74.5319,Y -45.9555,Z 89,A -153.7314,B 24.9244,C -2.0084,E1 24.8628,E2 238.7772} C_DIS
LIN {X -76.3514,Y -42.8621,Z 89,A -156.0265,B 24.9238,C -2.0162,E1 24.8596,E2 241.0656} C_DIS
LIN {X -78.7475,Y -38.2838,Z 89,A -159.3556,B 24.923,C -2.0269,E1 24.8554,E2 244.3869} C_DIS
LIN {X -80.4993,Y -34.4494,Z 89,A -162.2122,B 24.9226,C -2.0319,E1 24.8522,E2 247.2473} C_DIS
LIN {X -81.7591,Y -31.3406,Z 89,A -164.5225,B 24.9223,C -2.035,E1 24.8498,E2 249.5631} C_DIS
LIN {X -83.0617,Y -27.7036,Z 89,A -166.9244,B 24.9215,C -2.0461,E1 24.8476,E2 251.9524} C_DIS
LIN {X -84.0095,Y -24.6805,Z 89,A -168.8116,B 24.9206,C -2.0575,E1 24.8461,E2 253.823} C_DIS
LIN {X -84.9196,Y -21.3435,Z 89,A -171.3188,B 24.9206,C -2.0575,E1 24.8443,E2 256.3449} C_DIS
LIN {X -85.6323,Y -18.2737,Z 89,A -173.2012,B 24.9197,C -2.0689,E1 24.8431,E2 258.2112} C_DIS
LIN {X -86.4544,Y -13.876,Z 89,A -176.1325,B 24.919,C -2.0779,E1 24.8417,E2 261.1385} C_DIS
LIN {X -87.1683,Y -8.2708,Z 89,A 179.5298,B 24.9195,C -2.0716,E1 24.8403,E2 265.5172} C_DIS
LIN {X -87.5047,Y -3.1294,Z 89,A 175.7829,B 24.9195,C -2.0719,E1 24.8398,E2 269.2858} C_DIS
LIN {X -87.5549,Y 1.0361,Z 89,A 173.7986,B 24.9172,C -2.1012,E1 24.8398,E2 271.2121} C_DIS
LIN {X -87.1862,Y 8.0766,Z 89,A 167.849,B 24.9189,C -2.0791,E1 24.8411,E2 277.2502} C_DIS
LIN {X -86.4382,Y 13.9759,Z 89,A 165.4555,B 24.9147,C -2.1329,E1 24.842,E2 279.5295} C_DIS
LIN {X -85.4985,Y 18.8869,Z 89,A 161.7509,B 24.9148,C -2.1312,E1 24.844,E2 283.2602} C_DIS
LIN {X -84.5616,Y 22.7161,Z 89,A 159.5139,B 24.9134,C -2.1489,E1 24.8455,E2 285.4679} C_DIS
LIN {X -83.2826,Y 27.0309,Z 89,A 156.25,B 24.9134,C -2.1491,E1 24.8482,E2 288.7501} C_DIS
LIN {X -81.3815,Y 32.3082,Z 89,A 152.6224,B 24.9124,C -2.1615,E1 24.8518,E2 292.3685} C_DIS
LIN {X -80.2954,Y 34.9186,Z 89,A 150.9572,B 24.9115,C -2.1723,E1 24.8536,E2 294.0171} C_DIS
LIN {X -79.0932,Y 37.5644,Z 89,A 148.882,B 24.9115,C -2.1731,E1 24.856,E2 296.1018} C_DIS
LIN {X -77.5989,Y 40.5604,Z 89,A 147.0401,B 24.9101,C -2.1894,E1 24.8583,E2 297.9147} C_DIS
LIN {X -76.0466,Y 43.4009,Z 89,A 143.5728,B 24.9127,C -2.1577,E1 24.8632,E2 301.4758} C_DIS
LIN {X -73.4959,Y 47.5935,Z 89,A 141.3842,B 24.9096,C -2.1953,E1 24.8664,E2 303.5857} C_DIS
LIN {X -70.8359,Y 51.4683,Z 89,A 138.2406,B 24.9091,C -2.2018,E1 24.8714,E2 306.7294} C_DIS
LIN {X -67.1542,Y 56.1878,Z 89,A 134.2625,B 24.9084,C -2.2103,E1 24.8783,E2 310.7058} C_DIS
LIN {X -65.5413,Y 58.0621,Z 89,A 132.5097,B 24.9084,C -2.2105,E1 24.8815,E2 312.4659} C_DIS
LIN {X -62.8056,Y 61.0101,Z 89,A 129.9707,B 24.9076,C -2.2197,E1 24.8864,E2 314.9942} C_DIS
LIN {X -60.1192,Y 63.6583,Z 89,A 127.4858,B 24.9071,C -2.225,E1 24.8914,E2 317.4766} C_DIS
LIN {X -57.8724,Y 65.7083,Z 89,A 125.3845,B 24.9071,C -2.2263,E1 24.8958,E2 319.5832} C_DIS
LIN {X -54.8516,Y 68.2502,Z 89,A 122.7007,B 24.9068,C -2.2291,E1 24.9016,E2 322.2706} C_DIS
LIN {X -50.4995,Y 71.5308,Z 89,A 119.0983,B 24.9063,C -2.2353,E1 24.9097,E2 325.8708} C_DIS
LIN {X -46.5484,Y 74.1616,Z 89,A 115.9446,B 24.9059,C -2.2399,E1 24.9171,E2 329.0239} C_DIS
LIN {X -42.7442,Y 76.4173,Z 89,A 113.3073,B 24.9048,C -2.2525,E1 24.9234,E2 331.639} C_DIS
LIN {X -39.9393,Y 77.92,Z 89,A 111.3457,B 24.9042,C -2.2595,E1 24.9282,E2 333.5894} C_DIS
LIN {X -37.6964,Y 79.0298,Z 89,A 108.8146,B 24.9062,C -2.2358,E1 24.9348,E2 336.1833} C_DIS
LIN {X -33.8257,Y 80.7621,Z 89,A 106.9459,B 24.9036,C -2.2665,E1 24.9394,E2 337.9833} C_DIS
LIN {X -29.6539,Y 82.3859,Z 89,A 103.6543,B 24.9042,C -2.2595,E1 24.9481,E2 341.2983} C_DIS
LIN {X -25.7512,Y 83.6874,Z 89,A 101.3604,B 24.9029,C -2.2746,E1 24.9541,E2 343.5606} C_DIS
LIN {X -20.821,Y 85.0479,Z 89,A 98.2645,B 24.902,C -2.2856,E1 24.9624,E2 346.635} C_DIS
LIN {X -15.7147,Y 86.138,Z 89,A 94.4262,B 24.9028,C -2.2756,E1 24.9729,E2 350.5016} C_DIS
LIN {X -13.0147,Y 86.5876,Z 89,A 92.4201,B 24.9033,C -2.2703,E1 24.9785,E2 352.5221} C_DIS
LIN {X -8.3675,Y 87.1593,Z 89,A 88.7206,B 24.9048,C -2.2526,E1 24.9889,E2 356.2658} C_DIS
LIN {X -4.0259,Y 87.4673,Z 89,A 86.7071,B 24.9025,C -2.2792,E1 24.9943,E2 358.2168} C_DIS
LIN {X -0.7089,Y 87.5568,Z 89,A 83.9199,B 24.9041,C -2.2607,E1 25.0022,E2 361.0479} C_DIS
LIN {X 2.9308,Y 87.5108,Z 89,A 81.6557,B 24.9038,C -2.2646,E1 25.0085,E2 363.3024} C_DIS
LIN {X 6.1734,Y 87.342,Z 89,A 80.0167,B 24.9025,C -2.2796,E1 25.013,E2 364.905} C_DIS
LIN {X 9.8249,Y 87.0073,Z 89,A 76.9212,B 24.9044,C -2.2576,E1 25.0217,E2 368.0507} C_DIS
LIN {X 13.7226,Y 86.4782,Z 89,A 74.6209,B 24.9037,C -2.2653,E1 25.028,E2 370.3304} C_DIS
LIN {X 18.3563,Y 85.6143,Z 89,A 72.0405,B 24.9025,C -2.2799,E1 25.035,E2 372.8731} C_DIS
LIN {X 23.0796,Y 84.4633,Z 89,A 68.5922,B 24.9034,C -2.2695,E1 25.0444,E2 376.3408} C_DIS
LIN {X 27.1453,Y 83.2456,Z 89,A 66.0935,B 24.9028,C -2.2763,E1 25.051,E2 378.819} C_DIS
LIN {X 30.4371,Y 82.1003,Z 89,A 62.9278,B 24.9054,C -2.2459,E1 25.0594,E2 382.05} C_DIS
LIN {X 34.4434,Y 80.5018,Z 89,A 60.9242,B 24.9034,C -2.2692,E1 25.0645,E2 383.9937} C_DIS
LIN {X 36.6819,Y 79.5059,Z 89,A 59.2161,B 24.9038,C -2.264,E1 25.0688,E2 385.7099} C_DIS
LIN {X 40.4079,Y 77.679,Z 89,A 56.5542,B 24.904,C -2.2623,E1 25.0754,E2 388.3687} C_DIS
LIN {X 43.49,Y 75.9954,Z 89,A 54.3474,B 24.904,C -2.2621,E1 25.0808,E2 390.5694} C_DIS
LIN {X 48.6752,Y 72.7849,Z 89,A 50.2965,B 24.9047,C -2.254,E1 25.0904,E2 394.6266} C_DIS
LIN {X 51.1268,Y 71.0832,Z 89,A 47.758,B 24.9066,C -2.2314,E1 25.0962,E2 397.2095} C_DIS
LIN {X 54.118,Y 68.8328,Z 89,A 45.9476,B 24.9052,C -2.2481,E1 25.1001,E2 398.9738} C_DIS
LIN {X 56.2673,Y 67.088,Z 89,A 43.2239,B 24.908,C -2.2145,E1 25.1061,E2 401.7665} C_DIS
LIN {X 59.7852,Y 63.9724,Z 89,A 40.9427,B 24.9063,C -2.2345,E1 25.1107,E2 403.991} C_DIS
LIN {X 61.7159,Y 62.1118,Z 89,A 39.3199,B 24.9063,C -2.2352,E1 25.1139,E2 405.6053} C_DIS
LIN {X 65.6529,Y 57.9358,Z 89,A 35.5564,B 24.907,C -2.2267,E1 25.121,E2 409.3725} C_DIS
LIN {X 67.8459,Y 55.3505,Z 89,A 32.3623,B 24.9101,C -2.1888,E1 25.1268,E2 412.6413} C_DIS
LIN {X 70.9645,Y 51.2931,Z 89,A 29.9798,B 24.9081,C -2.213,E1 25.1306,E2 414.9552} C_DIS
LIN {X 72.7438,Y 48.7359,Z 89,A 27.6229,B 24.9095,C -2.197,E1 25.1343,E2 417.3381} C_DIS
LIN {X 75.2924,Y 44.696,Z 89,A 25.24,B 24.908,C -2.2142,E1 25.1378,E2 419.6684} C_DIS
LIN {X 76.7619,Y 42.1223,Z 89,A 22.6603,B 24.9103,C -2.1871,E1 25.1413,E2 422.2987} C_DIS
LIN {X 78.6577,Y 38.4681,Z 89,A 20.2739,B 24.91,C -2.1901,E1 25.1443,E2 424.6652} C_DIS
LIN {X 80.1312,Y 35.2954,Z 89,A 18.3518,B 24.9095,C -2.1963,E1 25.1465,E2 426.5624} C_DIS
LIN {X 81.5364,Y 31.9138,Z 89,A 15.696,B 24.9108,C -2.1804,E1 25.1493,E2 429.2409} C_DIS
LIN {X 82.606,Y 29.033,Z 89,A 13.2991,B 24.9124,C -2.1612,E1 25.1516,E2 431.6698} C_DIS
LIN {X 84.1386,Y 24.2347,Z 89,A 10.0332,B 24.9131,C -2.1523,E1 25.1543,E2 434.938} C_DIS
LIN {X 85.2718,Y 19.8851,Z 89,A 6.5927,B 24.9152,C -2.1262,E1 25.1565,E2 438.4202} C_DIS
LIN {X 86.1932,Y 15.4079,Z 89,A 3.9424,B 24.915,C -2.1286,E1 25.1578,E2 441.0494} C_DIS
LIN {X 86.7504,Y 11.8837,Z 89,A 2.1849,B 24.914,C -2.1412,E1 25.1585,E2 442.7668} C_DIS
LIN {X 87.1362,Y 8.6141,Z 89,A 0.2007,B 24.914,C -2.1403,E1 25.1591,E2 444.7413} C_DIS
LIN {X 87.4376,Y 4.6238,Z 89,A -2.992,B 24.9163,C -2.1121,E1 25.1597,E2 447.9817} C_DIS
LIN {X 87.5601,Y -0.1247,Z 89,A -5.6231,B 24.9158,C -2.1187,E1 25.1597,E2 450.5816} C_DIS
LIN {X 87.5193,Y -2.6523,Z 89,A -7.8854,B 24.9179,C -2.0923,E1 25.1596,E2 452.8927} C_DIS
LIN {X 87.3301,Y -6.3486,Z 89,A -10.0991,B 24.9179,C -2.0917,E1 25.1591,E2 455.0947} C_DIS
LIN {X 86.8684,Y -10.9822,Z 89,A -12.6645,B 24.9174,C -2.0987,E1 25.1584,E2 457.6284} C_DIS
LIN {X 86.398,Y -14.2162,Z 89,A -14.6039,B 24.9174,C -2.0988,E1 25.1575,E2 459.5561} C_DIS
LIN {X 85.6844,Y -18.0287,Z 89,A -17.5176,B 24.9191,C -2.0776,E1 25.156,E2 462.5029} C_DIS
LIN {X 84.5338,Y -22.8188,Z 89,A -20.0697,B 24.918,C -2.0909,E1 25.1543,E2 465.0088} C_DIS
LIN {X 83.4145,Y -26.6233,Z 89,A -23.8079,B 24.9217,C -2.043,E1 25.1512,E2 468.8388} C_DIS
LIN {X 82.1582,Y -30.2782,Z 89,A -25.6943,B 24.9206,C -2.0574,E1 25.1494,E2 470.6806} C_DIS
LIN {X 80.6055,Y -34.1966,Z 89,A -28.4259,B 24.9212,C -2.0499,E1 25.1465,E2 473.4148} C_DIS
LIN {X 79.1142,Y -37.5186,Z 89,A -30.9894,B 24.9222,C -2.0365,E1 25.1435,E2 475.9961} C_DIS
LIN {X 77.2945,Y -41.137,Z 89,A -33.5696,B 24.9226,C -2.0311,E1 25.1402,E2 478.5752} C_DIS
LIN {X 75.1905,Y -44.8686,Z 89,A -36.0842,B 24.9225,C -2.033,E1 25.1367,E2 481.0725} C_DIS
LIN {X 73.6962,Y -47.2814,Z 89,A -38.3437,B 24.9239,C -2.0139,E1 25.1333,E2 483.3656} C_DIS
LIN {X 69.65,Y -53.0638,Z 89,A -42.6584,B 24.9241,C -2.0117,E1 25.1263,E2 487.6647} C_DIS
LIN {X 65.9319,Y -57.6164,Z 89,A -45.9995,B 24.9236,C -2.0191,E1 25.1204,E2 490.9728} C_DIS
LIN {X 61.9215,Y -61.9085,Z 89,A -50.0745,B 24.9249,C -2.0015,E1 25.1126,E2 495.0717} C_DIS
LIN {X 58.2231,Y -65.3972,Z 89,A -53.2451,B 24.9251,C -1.999,E1 25.1061,E2 498.2352} C_DIS
LIN {X 54.1008,Y -68.8464,Z 89,A -56.9294,B 24.9261,C -1.9855,E1 25.0981,E2 501.9375} C_DIS
LIN {X 49.4773,Y -72.2418,Z 89,A -60.5899,B 24.9264,C -1.9808,E1 25.0899,E2 505.596} C_DIS
LIN {X 46.8843,Y -73.9502,Z 89,A -62.756,B 24.9271,C -1.9724,E1 25.0848,E2 507.7749} C_DIS
LIN {X 44.6401,Y -75.3255,Z 89,A -64.7848,B 24.9281,C -1.9589,E1 25.0798,E2 509.8293} C_DIS
LIN {X 39.842,Y -77.9697,Z 89,A -68.4956,B 24.9288,C -1.9487,E1 25.0707,E2 513.5539} C_DIS
LIN {X 34.9996,Y -80.2601,Z 89,A -71.8198,B 24.9288,C -1.9493,E1 25.0622,E2 516.8683} C_DIS
LIN {X 31.2159,Y -81.8063,Z 89,A -74.6754,B 24.9295,C -1.9396,E1 25.0548,E2 519.7405} C_DIS
LIN {X 26.8254,Y -83.3491,Z 89,A -78.1059,B 24.9306,C -1.9233,E1 25.0456,E2 523.203} C_DIS
LIN {X 22.7495,Y -84.5525,Z 89,A -79.8091,B 24.9283,C -1.9555,E1 25.0412,E2 524.8272} C_DIS
LIN {X 18.5522,Y -85.5715,Z 89,A -82.6101,B 24.9284,C -1.9536,E1 25.0336,E2 527.6288} C_DIS
LIN {X 14.2415,Y -86.3938,Z 89,A -85.8369,B 24.9295,C -1.9397,E1 25.0247,E2 530.8849} C_DIS
LIN {X 10.8476,Y -86.8859,Z 89,A -88.0499,B 24.9295,C -1.9392,E1 25.0185,E2 533.0971} C_DIS
LIN {X 7.7187,Y -87.2192,Z 89,A -90.1111,B 24.9295,C -1.938,E1 25.0128,E2 535.1599} C_DIS
LIN {X 4.8679,Y -87.4241,Z 89,A -92.3782,B 24.9306,C -1.9246,E1 25.0064,E2 537.458} C_DIS
LIN {X 0.5712,Y -87.548,Z 89,A -94.3117,B 24.9286,C -1.952,E1 25.0012,E2 539.3261} C_DIS
Enddeposition()
LIN {X 0.5712,Y -87.548,Z 89,A -94.3117,B 24.9286,C -1.952,E1 25.0012,E2 539.3261} C_DIS
Startdeposition()
$VEL.CP = VEL_PRINT
LIN {X 1.0911,Y -86.5597,Z 89,A -92.7469,B 24.9244,C -2.0085,E1 25.006,E2 537.6275} C_DIS
LIN {X 4.9782,Y -86.4232,Z 89,A -90.967,B 24.9262,C -1.9838,E1 25.0107,E2 535.9069} C_DIS
LIN {X 7.8637,Y -86.2084,Z 89,A -89.0342,B 24.9262,C -1.9853,E1 25.0161,E2 533.9716} C_DIS
LIN {X 10.9726,Y -85.8682,Z 89,A -86.9017,B 24.9259,C -1.9886,E1 25.022,E2 531.8328} C_DIS
LIN {X 16.0396,Y -85.0676,Z 89,A -83.517,B 24.9257,C -1.9908,E1 25.0314,E2 528.4464} C_DIS
LIN {X 19.7484,Y -84.284,Z 89,A -81.1889,B 24.926,C -1.9871,E1 25.0377,E2 526.13} C_DIS
LIN {X 22.3954,Y -83.6194,Z 89,A -79.2033,B 24.9254,C -1.9949,E1 25.0431,E2 524.1291} C_DIS
LIN {X 26.572,Y -82.3872,Z 89,A -76.0128,B 24.9244,C -2.0084,E1 25.0517,E2 520.9122} C_DIS
LIN {X 30.9614,Y -80.8407,Z 89,A -73.4784,B 24.9254,C -1.9943,E1 25.0582,E2 518.4166} C_DIS
LIN {X 32.9893,Y -80.0348,Z 89,A -71.7992,B 24.9247,C -2.0042,E1 25.0626,E2 516.7178} C_DIS
LIN {X 37.6556,Y -77.9475,Z 89,A -68.7324,B 24.9251,C -1.9988,E1 25.0704,E2 513.6714} C_DIS
LIN {X 39.541,Y -77.0081,Z 89,A -67.011,B 24.9241,C -2.0121,E1 25.0747,E2 511.9234} C_DIS
LIN {X 42.6108,Y -75.3537,Z 89,A -64.7415,B 24.9239,C -2.0148,E1 25.0803,E2 509.654} C_DIS
LIN {X 47.1322,Y -72.6117,Z 89,A -61.2233,B 24.9233,C -2.022,E1 25.0886,E2 506.13} C_DIS
LIN {X 50.9624,Y -69.9757,Z 89,A -58.0248,B 24.9226,C -2.0323,E1 25.096,E2 502.9181} C_DIS
LIN {X 54.2138,Y -67.4887,Z 89,A -55.7673,B 24.9233,C -2.0227,E1 25.1009,E2 500.6915} C_DIS
LIN {X 57.0689,Y -65.0914,Z 89,A -53.3156,B 24.9229,C -2.0277,E1 25.1061,E2 498.2376} C_DIS
LIN {X 60.144,Y -62.2609,Z 89,A -50.4653,B 24.9222,C -2.0371,E1 25.1119,E2 495.3768} C_DIS
LIN {X 62.0823,Y -60.3293,Z 89,A -47.7641,B 24.9195,C -2.0722,E1 25.1173,E2 492.6041} C_DIS
LIN {X 64.8216,Y -57.3769,Z 89,A -46.0238,B 24.9214,C -2.0469,E1 25.1205,E2 490.9314} C_DIS
LIN {X 67.0884,Y -54.7077,Z 89,A -43.6823,B 24.9209,C -2.0538,E1 25.1247,E2 488.5844} C_DIS
LIN {X 68.7795,Y -52.5663,Z 89,A -41.5975,B 24.9198,C -2.0682,E1 25.1283,E2 486.4754} C_DIS
LIN {X 71.3992,Y -48.9502,Z 89,A -38.7319,B 24.9194,C -2.0732,E1 25.1329,E2 483.612} C_DIS
LIN {X 74.4321,Y -44.1996,Z 89,A -35.482,B 24.9199,C -2.0671,E1 25.1377,E2 480.3929} C_DIS
LIN {X 76.7042,Y -40.1278,Z 89,A -32.4812,B 24.9194,C -2.073,E1 25.1418,E2 477.3937} C_DIS
LIN {X 78.2769,Y -36.9686,Z 89,A -29.317,B 24.9166,C -2.1088,E1 25.1457,E2 474.1619} C_DIS
LIN {X 80.4751,Y -31.8991,Z 89,A -26.4052,B 24.9178,C -2.0939,E1 25.1488,E2 471.3014} C_DIS
LIN {X 81.316,Y -29.6889,Z 89,A -23.4889,B 24.9136,C -2.1463,E1 25.1517,E2 468.2778} C_DIS
LIN {X 82.8989,Y -24.9317,Z 89,A -21.1805,B 24.9156,C -2.1209,E1 25.1535,E2 466.0424} C_DIS
LIN {X 83.7924,Y -21.739,Z 89,A -19.0457,B 24.9153,C -2.1257,E1 25.1551,E2 463.9085} C_DIS
LIN {X 84.6598,Y -18.0716,Z 89,A -15.9342,B 24.9129,C -2.1554,E1 25.157,E2 460.7452} C_DIS
LIN {X 85.3474,Y -14.4769,Z 89,A -14.1344,B 24.914,C -2.1412,E1 25.1578,E2 458.9894} C_DIS
LIN {X 85.7778,Y -11.6683,Z 89,A -12.1512,B 24.9132,C -2.1507,E1 25.1586,E2 456.9953} C_DIS
Enddeposition()
END
